C07239=1059.331,223.507,-90.302,172.650,33.223,156.173
C07240=1059.324,223.257,-90.275,172.647,33.219,156.173
C07241=1059.319,223.009,-90.249,172.645,33.215,156.172
C07242=1059.313,222.761,-90.222,172.642,33.212,156.171
C07243=1059.307,222.526,-90.196,172.640,33.208,156.170
C07244=1059.300,222.291,-90.172,172.638,33.204,156.170
C07245=1059.295,222.056,-90.147,172.637,33.201,156.169
C07246=1059.289,221.821,-90.121,172.635,33.197,156.168
C07247=1059.283,221.586,-90.096,172.633,33.193,156.168
C07248=1059.278,221.351,-90.071,172.631,33.190,156.167
C07249=1059.272,221.116,-90.045,172.629,33.185,156.166
C07250=1059.266,220.881,-90.020,172.627,33.182,156.166
C07251=1059.260,220.633,-89.994,172.625,33.178,156.165
C07252=1059.254,220.384,-89.968,172.623,33.174,156.164
C07253=1059.247,220.135,-89.942,172.621,33.171,156.163
C07254=1059.241,219.887,-89.915,172.619,33.166,156.163
C07255=1059.235,219.639,-89.889,172.617,33.163,156.162
C07256=1059.229,219.390,-89.862,172.615,33.159,156.161
C07257=1059.222,219.141,-89.837,172.613,33.155,156.160
C07258=1059.216,218.893,-89.810,172.611,33.151,156.160
C07259=1059.211,218.644,-89.783,172.609,33.147,156.159
C07260=1059.204,218.396,-89.757,172.607,33.143,156.158
C07261=1059.198,218.147,-89.730,172.604,33.140,156.158
C07262=1059.191,217.898,-89.705,172.602,33.135,156.157
C07263=1059.186,217.650,-89.678,172.600,33.132,156.156
C07264=1059.179,217.402,-89.652,172.598,33.128,156.155
C07265=1059.173,217.152,-89.626,172.596,33.124,156.155
C07266=1059.167,216.904,-89.600,172.594,33.120,156.154
C07267=1059.161,216.656,-89.573,172.592,33.116,156.153
C07268=1059.155,216.407,-89.548,172.590,33.112,156.152
C07269=1059.149,216.159,-89.521,172.588,33.108,156.152
C07270=1059.142,215.910,-89.495,172.586,33.104,156.151
C07271=1059.136,215.661,-89.469,172.584,33.101,156.150
C07272=1059.130,215.413,-89.443,172.582,33.096,156.149
C07273=1059.124,215.165,-89.416,172.580,33.093,156.149
C07274=1059.118,214.916,-89.391,172.578,33.088,156.148
C07275=1059.111,214.667,-89.364,172.576,33.085,156.147
C07276=1059.105,214.418,-89.339,172.574,33.080,156.146
C07277=1059.099,214.170,-89.312,172.573,33.077,156.146
C07278=1059.093,213.921,-89.287,172.571,33.073,156.145
C07279=1059.087,213.673,-89.260,172.568,33.069,156.144
C07280=1059.081,213.425,-89.234,172.566,33.065,156.144
C07281=1059.075,213.176,-89.208,172.564,33.061,156.143
C07282=1059.069,212.928,-89.182,172.562,33.057,156.142
C07283=1059.063,212.678,-89.156,172.560,33.053,156.141
C07284=1059.056,212.430,-89.130,172.558,33.049,156.141
C07285=1059.050,212.181,-89.104,172.556,33.045,156.140
C07286=1059.045,211.932,-89.078,172.554,33.041,156.139
C07287=1059.038,211.684,-89.052,172.552,33.037,156.138
C07288=1059.032,211.436,-89.027,172.550,33.033,156.138
C07289=1059.026,211.187,-89.000,172.548,33.029,156.137
C07290=1059.020,210.939,-88.975,172.546,33.026,156.136
C07291=1059.013,210.690,-88.949,172.544,33.022,156.135
C07292=1059.007,210.441,-88.923,172.542,33.018,156.135
C07293=1059.001,210.192,-88.897,172.540,33.014,156.134
C07294=1058.995,209.944,-88.871,172.538,33.010,156.133
C07295=1058.988,209.696,-88.846,172.536,33.006,156.132
C07296=1058.983,209.447,-88.820,172.534,33.002,156.132
C07297=1058.976,209.199,-88.794,172.532,32.998,156.131
C07298=1058.970,208.950,-88.769,172.530,32.994,156.130
C07299=1058.965,208.717,-88.744,172.529,32.990,156.130
C07300=1058.959,208.484,-88.720,172.527,32.986,156.129
C07301=1058.954,208.252,-88.696,172.525,32.983,156.128
C07302=1058.947,208.020,-88.672,172.523,32.979,156.127
C07303=1058.941,207.788,-88.648,172.521,32.975,156.127
C07304=1058.936,207.555,-88.624,172.520,32.972,156.126
C07305=1058.930,207.323,-88.600,172.518,32.968,156.125
C07306=1058.924,207.090,-88.576,172.516,32.964,156.125
C07307=1058.899,206.041,-88.472,172.330,32.878,156.114
C07308=1058.893,205.792,-88.447,172.327,32.874,156.114
C07309=1058.888,205.543,-88.423,172.325,32.871,156.113
C07310=1058.881,205.295,-88.398,172.323,32.868,156.113
C07311=1058.875,205.045,-88.373,172.320,32.865,156.112
C07312=1058.870,204.797,-88.348,172.318,32.862,156.112
C07313=1058.864,204.548,-88.323,172.316,32.859,156.111
C07314=1058.858,204.300,-88.298,172.313,32.856,156.110
C07315=1058.852,204.051,-88.274,172.311,32.853,156.110
C07316=1058.846,203.802,-88.250,172.309,32.850,156.109
C07317=1058.840,203.554,-88.225,172.306,32.846,156.109
C07318=1058.834,203.304,-88.200,172.304,32.843,156.108
C07319=1058.829,203.056,-88.176,172.302,32.841,156.108
C07320=1058.823,202.807,-88.151,172.299,32.838,156.107
C07321=1058.817,202.559,-88.126,172.297,32.834,156.107
C07322=1058.811,202.310,-88.102,172.295,32.831,156.106
C07323=1058.805,202.062,-88.077,172.292,32.828,156.106
C07324=1058.799,201.812,-88.053,172.290,32.825,156.105
C07325=1058.793,201.563,-88.028,172.288,32.822,156.105
C07326=1058.787,201.315,-88.004,172.285,32.819,156.104
C07327=1058.781,201.066,-87.980,172.283,32.816,156.104
C07328=1058.775,200.818,-87.955,172.281,32.813,156.103
C07329=1058.769,200.569,-87.931,172.278,32.810,156.103
C07330=1058.763,200.320,-87.907,172.276,32.807,156.102
C07331=1058.757,200.071,-87.883,172.274,32.804,156.102
C07332=1058.751,199.822,-87.858,172.271,32.801,156.101
C07333=1058.745,199.573,-87.834,172.269,32.798,156.100
C07334=1058.739,199.325,-87.809,172.267,32.796,156.100
C07335=1058.733,199.077,-87.785,172.265,32.792,156.099
C07336=1058.727,198.827,-87.761,172.262,32.789,156.099
C07337=1058.721,198.579,-87.737,172.260,32.787,156.098
C07338=1058.715,198.330,-87.712,172.258,32.783,156.098
C07339=1058.709,198.081,-87.689,172.255,32.780,156.097
C07340=1058.703,197.832,-87.664,172.253,32.778,156.097
C07341=1058.697,197.584,-87.640,172.251,32.775,156.096
C07342=1058.691,197.335,-87.616,172.248,32.771,156.096
C07343=1058.685,197.086,-87.592,172.247,32.769,156.095
C07344=1058.679,196.837,-87.568,172.245,32.766,156.095
C07345=1058.674,196.588,-87.543,172.243,32.762,156.094
C07346=1058.668,196.339,-87.519,172.240,32.760,156.094
C07347=1058.662,196.091,-87.495,172.238,32.757,156.093
C07348=1058.656,195.843,-87.471,172.236,32.754,156.093
C07349=1058.650,195.593,-87.447,172.234,32.751,156.092
C07350=1058.644,195.345,-87.423,172.231,32.748,156.092
C07351=1058.638,195.096,-87.398,172.229,32.745,156.091
C07352=1058.632,194.847,-87.375,172.227,32.742,156.091
C07353=1058.626,194.598,-87.350,172.224,32.739,156.090
C07354=1058.620,194.350,-87.326,172.222,32.736,156.090
C07355=1058.615,194.101,-87.302,172.220,32.733,156.089
C07356=1058.608,193.852,-87.278,172.218,32.730,156.089
C07357=1058.603,193.604,-87.254,172.215,32.727,156.088
C07358=1058.597,193.355,-87.230,172.213,32.724,156.088
C07359=1058.592,193.106,-87.206,172.211,32.722,156.087
C07360=1058.586,192.857,-87.183,172.209,32.718,156.087
C07361=1058.579,192.608,-87.159,172.207,32.715,156.086
C07362=1058.574,192.360,-87.134,172.204,32.713,156.086
C07363=1058.568,192.111,-87.111,172.202,32.709,156.085
C07364=1058.562,191.862,-87.086,172.200,32.707,156.085
C07365=1058.556,191.613,-87.063,172.198,32.704,156.084
C07366=1058.551,191.365,-87.039,172.195,32.700,156.084
C07367=1058.544,191.116,-87.015,172.193,32.698,156.083
C07368=1058.538,190.832,-86.988,172.191,32.695,156.083
C07369=1058.531,190.548,-86.960,172.188,32.691,156.082
C07370=1058.525,190.265,-86.934,172.186,32.688,156.081
C07371=1058.518,189.981,-86.906,172.184,32.684,156.081
C07372=1058.511,189.732,-86.882,172.182,32.681,156.080
C07373=1058.507,189.483,-86.858,172.180,32.679,156.080
C07374=1058.500,189.235,-86.835,172.177,32.675,156.079
C07375=1058.494,188.986,-86.811,172.175,32.672,156.079
C07376=1058.489,188.736,-86.787,172.173,32.670,156.078
C07377=1058.483,188.488,-86.763,172.171,32.667,156.078
C07378=1058.478,188.240,-86.739,172.169,32.664,156.077
C07379=1058.471,187.990,-86.716,172.166,32.661,156.077
C07380=1058.466,187.741,-86.692,172.164,32.658,156.076
C07381=1058.460,187.493,-86.668,172.162,32.655,156.076
C07382=1058.454,187.244,-86.645,172.160,32.652,156.075
C07383=1058.449,186.996,-86.621,172.158,32.649,156.075
C07384=1058.442,186.746,-86.597,172.156,32.646,156.074
C07385=1058.437,186.497,-86.573,172.153,32.644,156.074
C07386=1058.431,186.249,-86.550,172.151,32.640,156.073
C07387=1058.425,186.000,-86.527,172.149,32.638,156.073
C07388=1058.420,185.752,-86.502,172.147,32.635,156.072
C07389=1058.414,185.502,-86.479,172.145,32.631,156.072
C07390=1058.408,185.253,-86.455,172.143,32.629,156.071
C07391=1058.403,185.005,-86.432,172.140,32.626,156.071
C07392=1058.397,184.756,-86.408,172.138,32.623,156.070
C07393=1058.392,184.507,-86.385,172.136,32.620,156.070
C07394=1058.385,184.258,-86.361,172.134,32.617,156.069
C07395=1058.379,184.009,-86.338,172.133,32.614,156.069
C07396=1058.373,183.761,-86.314,172.131,32.612,156.068
C07397=1058.367,183.511,-86.291,172.128,32.609,156.068
C07398=1058.361,183.262,-86.268,172.126,32.606,156.068
C07399=1058.355,183.014,-86.244,172.124,32.603,156.067
C07400=1058.349,182.765,-86.221,172.122,32.601,156.067
C07401=1058.343,182.516,-86.198,172.120,32.598,156.066
C07402=1058.336,182.268,-86.175,172.118,32.595,156.066
C07403=1058.331,182.019,-86.152,172.115,32.592,156.065
C07404=1058.325,181.770,-86.129,172.113,32.590,156.065
C07405=1058.318,181.521,-86.105,172.111,32.587,156.064
C07406=1058.313,181.272,-86.082,172.109,32.584,156.064
C07407=1058.307,181.023,-86.059,172.107,32.581,156.063
C07408=1058.301,180.775,-86.035,172.105,32.579,156.063
C07409=1058.294,180.525,-86.012,172.102,32.576,156.063
C07410=1058.289,180.276,-85.989,172.100,32.573,156.062
C07411=1058.283,180.027,-85.966,172.098,32.570,156.062
C07412=1058.276,179.779,-85.943,172.096,32.568,156.061
C07413=1058.270,179.531,-85.920,172.094,32.565,156.061
C07414=1058.264,179.281,-85.897,172.092,32.562,156.060
C07415=1058.258,179.032,-85.874,172.090,32.559,156.060
C07416=1058.252,178.784,-85.850,172.088,32.557,156.059
C07417=1058.247,178.535,-85.827,172.086,32.554,156.059
C07418=1058.241,178.286,-85.804,172.084,32.551,156.058
C07419=1058.235,178.037,-85.781,172.082,32.548,156.058
C07420=1058.228,177.788,-85.759,172.080,32.546,156.057
C07421=1058.222,177.539,-85.736,172.078,32.543,156.057
C07422=1058.216,177.291,-85.712,172.076,32.540,156.056
C07423=1058.211,177.042,-85.689,172.073,32.537,156.056
C07424=1058.205,176.793,-85.666,172.071,32.535,156.056
C07425=1058.199,176.544,-85.643,172.069,32.532,156.055
C07426=1058.193,176.295,-85.620,172.067,32.529,156.055
C07427=1058.186,176.046,-85.597,172.065,32.527,156.054
C07428=1058.181,175.797,-85.574,172.063,32.524,156.054
C07429=1058.175,175.548,-85.552,172.061,32.521,156.053
C07430=1058.169,175.299,-85.529,172.059,32.518,156.053
C07431=1058.163,175.050,-85.506,172.057,32.516,156.052
C07432=1058.156,174.766,-85.479,172.054,32.512,156.052
C07433=1058.149,174.482,-85.454,172.052,32.509,156.051
C07434=1058.143,174.198,-85.427,172.050,32.506,156.051
C07435=1058.137,173.914,-85.401,172.048,32.503,156.050
C07436=1058.131,173.665,-85.378,172.046,32.500,156.050
C07437=1058.125,173.416,-85.355,172.044,32.498,156.049
C07438=1058.118,173.167,-85.333,172.042,32.495,156.049
C07439=1058.112,172.918,-85.310,172.040,32.492,156.048
C07440=1058.107,172.669,-85.287,172.038,32.489,156.048
C07441=1058.101,172.420,-85.264,172.036,32.487,156.047
C07442=1058.095,172.171,-85.241,172.034,32.483,156.047
C07443=1058.089,171.923,-85.219,172.031,32.481,156.047
C07444=1058.083,171.674,-85.196,172.029,32.478,156.046
C07445=1058.077,171.425,-85.173,172.027,32.476,156.046
C07446=1058.071,171.176,-85.150,172.025,32.472,156.045
C07447=1058.066,170.927,-85.127,172.023,32.470,156.045
C07448=1058.059,170.679,-85.104,172.021,32.467,156.044
C07449=1058.054,170.429,-85.082,172.019,32.465,156.044
C07450=1058.048,170.180,-85.059,172.017,32.461,156.043
C07451=1058.042,169.931,-85.036,172.015,32.459,156.043
C07452=1058.037,169.682,-85.013,172.014,32.456,156.042
C07453=1058.031,169.435,-84.991,172.012,32.454,156.042
C07454=1058.025,169.186,-84.968,172.010,32.451,156.041
C07455=1058.020,168.936,-84.946,172.008,32.448,156.041
C07456=1058.014,168.687,-84.923,172.006,32.445,156.041
C07457=1058.007,168.439,-84.901,172.004,32.443,156.040
C07458=1058.002,168.190,-84.878,172.002,32.440,156.040
C07459=1057.996,167.941,-84.855,172.000,32.437,156.039
C07460=1057.991,167.691,-84.833,171.998,32.434,156.039
C07461=1057.985,167.442,-84.810,171.996,32.432,156.038
C07462=1057.978,167.194,-84.787,171.994,32.429,156.038
C07463=1057.973,166.945,-84.765,171.992,32.426,156.037
C07464=1057.967,166.695,-84.742,171.989,32.423,156.037
C07465=1057.962,166.447,-84.720,171.987,32.421,156.036
C07466=1057.956,166.199,-84.697,171.985,32.418,156.036
C07467=1057.950,165.949,-84.675,171.983,32.415,156.036
C07468=1057.944,165.700,-84.652,171.982,32.412,156.035
C07469=1057.938,165.452,-84.630,171.980,32.410,156.035
C07470=1057.933,165.202,-84.608,171.978,32.407,156.034
C07471=1057.927,164.953,-84.585,171.976,32.404,156.034
C07472=1057.921,164.704,-84.562,171.974,32.401,156.033
C07473=1057.916,164.456,-84.540,171.972,32.399,156.033
C07474=1057.910,164.207,-84.517,171.970,32.396,156.032
C07475=1057.904,163.958,-84.495,171.968,32.393,156.032
C07476=1057.899,163.709,-84.472,171.966,32.391,156.031
C07477=1057.892,163.460,-84.450,171.964,32.388,156.031
C07478=1057.887,163.212,-84.427,171.962,32.385,156.030
C07479=1057.882,162.962,-84.405,171.960,32.382,156.030
C07480=1057.875,162.714,-84.383,171.958,32.380,156.030
C07481=1057.870,162.464,-84.361,171.956,32.376,156.029
C07482=1057.864,162.215,-84.338,171.954,32.374,156.029
C07483=1057.859,161.966,-84.316,171.952,32.371,156.028
C07484=1057.853,161.718,-84.293,171.952,32.369,156.028
C07485=1057.847,161.468,-84.271,171.950,32.366,156.027
C07486=1057.842,161.219,-84.248,171.948,32.363,156.027
C07487=1057.835,160.970,-84.227,171.946,32.360,156.026
C07488=1057.830,160.722,-84.204,171.944,32.358,156.026
C07489=1057.824,160.473,-84.182,171.942,32.355,156.025
C07490=1057.818,160.224,-84.159,171.940,32.353,156.025
C07491=1057.812,159.975,-84.138,171.938,32.350,156.025
C07492=1057.806,159.726,-84.115,171.936,32.347,156.024
C07493=1057.800,159.477,-84.093,171.934,32.344,156.024
C07494=1057.795,159.228,-84.072,171.932,32.342,156.023
C07495=1057.788,158.980,-84.050,171.930,32.339,156.023
C07496=1057.782,158.694,-84.025,171.927,32.336,156.022
C07497=1057.775,158.410,-83.999,171.925,32.333,156.022
C07498=1057.768,158.126,-83.973,171.924,32.330,156.021
C07499=1057.762,157.841,-83.949,171.922,32.327,156.021
C07500=1057.756,157.592,-83.927,171.920,32.325,156.020
C07501=1057.749,157.343,-83.905,171.918,32.322,156.020
C07502=1057.744,157.094,-83.882,171.916,32.319,156.020
C07503=1057.738,156.845,-83.861,171.914,32.317,156.019
C07504=1057.732,156.597,-83.839,171.912,32.314,156.019
C07505=1057.726,156.347,-83.817,171.910,32.311,156.018
C07506=1057.720,156.098,-83.795,171.908,32.309,156.018
C07507=1057.714,155.849,-83.773,171.906,32.306,156.017
C07508=1057.709,155.601,-83.751,171.904,32.303,156.017
C07509=1057.703,155.351,-83.729,171.902,32.301,156.016
C07510=1057.697,155.102,-83.707,171.900,32.298,156.016
C07511=1057.691,154.853,-83.686,171.898,32.296,156.016
C07512=1057.685,154.605,-83.663,171.897,32.293,156.015
C07513=1057.679,154.356,-83.642,171.895,32.290,156.015
C07514=1057.673,154.106,-83.620,171.893,32.288,156.014
C07515=1057.667,153.857,-83.598,171.891,32.285,156.014
C07516=1057.661,153.609,-83.577,171.889,32.282,156.013
C07517=1057.656,153.360,-83.554,171.887,32.280,156.013
C07518=1057.649,153.111,-83.533,171.885,32.277,156.013
C07519=1057.643,152.861,-83.511,171.883,32.275,156.012
C07520=1057.638,152.613,-83.490,171.882,32.272,156.012
C07521=1057.632,152.364,-83.468,171.880,32.270,156.011
C07522=1057.625,152.114,-83.446,171.878,32.267,156.011
C07523=1057.620,151.865,-83.424,171.876,32.264,156.010
C07524=1057.614,151.616,-83.403,171.874,32.262,156.010
C07525=1057.608,151.368,-83.380,171.872,32.259,156.010
C07526=1057.602,151.119,-83.359,171.871,32.257,156.009
C07527=1057.596,150.870,-83.338,171.869,32.254,156.009
C07528=1057.590,150.621,-83.316,171.867,32.251,156.008
C07529=1057.585,150.371,-83.294,171.865,32.249,156.008
C07530=1057.579,150.123,-83.272,171.863,32.246,156.007
C07531=1057.573,149.874,-83.251,171.861,32.244,156.007
C07532=1057.567,149.625,-83.229,171.859,32.241,156.007
C07533=1057.561,149.376,-83.208,171.857,32.238,156.006
C07534=1057.555,149.127,-83.186,171.856,32.236,156.006
C07535=1057.549,148.878,-83.165,171.854,32.233,156.005
C07536=1057.543,148.629,-83.143,171.852,32.231,156.005
C07537=1057.537,148.380,-83.122,171.850,32.228,156.004
C07538=1057.531,148.131,-83.100,171.848,32.225,156.004
C07539=1057.526,147.882,-83.078,171.846,32.223,156.004
C07540=1057.520,147.633,-83.057,171.845,32.220,156.003
C07541=1057.514,147.383,-83.035,171.843,32.218,156.003
C07542=1057.508,147.135,-83.014,171.841,32.215,156.002
C07543=1057.502,146.885,-82.993,171.839,32.212,156.002
C07544=1057.495,146.636,-82.972,171.837,32.210,156.002
C07545=1057.490,146.388,-82.950,171.835,32.207,156.001
C07546=1057.484,146.139,-82.929,171.834,32.205,156.001
C07547=1057.478,145.890,-82.908,171.832,32.202,156.000
C07548=1057.472,145.641,-82.886,171.830,32.199,156.000
C07549=1057.466,145.392,-82.864,171.828,32.197,155.999
C07550=1057.460,145.143,-82.843,171.826,32.195,155.999
C07551=1057.454,144.893,-82.822,171.824,32.192,155.999
C07552=1057.448,144.644,-82.800,171.823,32.190,155.998
C07553=1057.443,144.396,-82.779,171.821,32.187,155.998
C07554=1057.437,144.146,-82.758,171.819,32.184,155.997
C07555=1057.431,143.898,-82.736,171.817,32.182,155.997
C07556=1057.424,143.648,-82.716,171.816,32.179,155.997
C07557=1057.418,143.399,-82.694,171.814,32.177,155.996
C07558=1057.413,143.151,-82.673,171.812,32.174,155.996
C07559=1057.407,142.901,-82.651,171.810,32.171,155.995
C07560=1057.401,142.616,-82.628,171.808,32.169,155.995
C07561=1057.394,142.332,-82.603,171.806,32.166,155.994
C07562=1057.386,142.047,-82.579,171.803,32.163,155.994
C07563=1057.380,141.763,-82.554,171.801,32.160,155.993
C07564=1057.374,141.513,-82.533,171.800,32.157,155.993
C07565=1057.368,141.265,-82.513,171.799,32.155,155.992
C07566=1057.362,141.015,-82.491,171.797,32.152,155.992
C07567=1057.356,140.766,-82.470,171.795,32.149,155.992
C07568=1057.351,140.517,-82.449,171.793,32.147,155.991
C07569=1057.344,140.268,-82.427,171.791,32.144,155.991
C07570=1057.339,140.019,-82.407,171.789,32.142,155.990
C07571=1057.333,139.769,-82.385,171.787,32.139,155.990
C07572=1057.327,139.521,-82.364,171.786,32.137,155.990
C07573=1057.321,139.271,-82.343,171.784,32.134,155.989
C07574=1057.315,139.023,-82.322,171.782,32.132,155.989
C07575=1057.309,138.773,-82.301,171.780,32.129,155.988
C07576=1057.303,138.525,-82.281,171.778,32.126,155.988
C07577=1057.297,138.276,-82.259,171.777,32.124,155.987
C07578=1057.292,138.027,-82.238,171.775,32.121,155.987
C07579=1057.285,137.777,-82.217,171.773,32.119,155.987
C07580=1057.279,137.529,-82.197,171.772,32.117,155.986
C07581=1057.273,137.279,-82.175,171.770,32.114,155.986
C07582=1057.268,137.030,-82.155,171.768,32.111,155.985
C07583=1057.261,136.781,-82.133,171.766,32.109,155.985
C07584=1057.256,136.532,-82.113,171.764,32.106,155.985
C07585=1057.250,136.283,-82.091,171.762,32.104,155.984
C07586=1057.244,136.034,-82.071,171.760,32.102,155.984
C07587=1057.238,135.785,-82.050,171.759,32.099,155.983
C07588=1057.232,135.536,-82.029,171.757,32.096,155.983
C07589=1057.225,135.287,-82.008,171.756,32.094,155.983
C07590=1057.220,135.038,-81.988,171.754,32.091,155.982
C07591=1057.214,134.789,-81.966,171.752,32.089,155.982
C07592=1057.208,134.540,-81.946,171.750,32.086,155.981
C07593=1057.202,134.291,-81.924,171.749,32.084,155.981
C07594=1057.196,134.042,-81.904,171.747,32.081,155.981
C07595=1057.190,133.792,-81.883,171.745,32.079,155.980
C07596=1057.184,133.543,-81.862,171.743,32.076,155.980
C07597=1057.178,133.295,-81.842,171.741,32.074,155.979
C07598=1057.172,133.045,-81.821,171.739,32.071,155.979
C07599=1057.167,132.796,-81.800,171.738,32.068,155.978
C07600=1057.160,132.547,-81.780,171.737,32.066,155.978
C07601=1057.155,132.298,-81.758,171.735,32.063,155.978
C07602=1057.149,132.050,-81.738,171.733,32.061,155.977
C07603=1057.143,131.800,-81.718,171.731,32.059,155.977
C07604=1057.137,131.551,-81.696,171.729,32.056,155.976
C07605=1057.131,131.302,-81.676,171.728,32.053,155.976
C07606=1057.125,131.053,-81.656,171.726,32.051,155.976
C07607=1057.119,130.804,-81.634,171.724,32.049,155.975
C07608=1057.113,130.555,-81.614,171.722,32.046,155.975
C07609=1057.106,130.305,-81.594,171.720,32.044,155.974
C07610=1057.101,130.056,-81.574,171.718,32.041,155.974
C07611=1057.094,129.807,-81.552,171.717,32.039,155.974
C07612=1057.089,129.558,-81.532,171.716,32.036,155.973
C07613=1057.083,129.309,-81.512,171.714,32.034,155.973
C07614=1057.076,129.060,-81.492,171.712,32.031,155.972
C07615=1057.071,128.811,-81.470,171.710,32.029,155.972
C07616=1057.064,128.562,-81.450,171.708,32.026,155.972
C07617=1057.058,128.313,-81.430,171.707,32.024,155.971
C07618=1057.053,128.064,-81.410,171.705,32.021,155.971
C07619=1057.046,127.814,-81.389,171.703,32.019,155.971
C07620=1057.040,127.566,-81.369,171.701,32.017,155.970
C07621=1057.034,127.316,-81.348,171.699,32.014,155.970
C07622=1057.028,127.068,-81.328,171.698,32.012,155.969
C07623=1057.022,126.819,-81.308,171.697,32.010,155.969
C07624=1057.015,126.533,-81.284,171.695,32.006,155.968
C07625=1057.009,126.249,-81.261,171.693,32.004,155.968
C07626=1057.002,125.963,-81.237,171.690,32.001,155.968
C07627=1056.994,125.679,-81.214,171.688,31.998,155.967
C07628=1056.989,125.429,-81.194,171.687,31.996,155.967
C07629=1056.983,125.180,-81.174,171.685,31.993,155.966
C07630=1056.977,124.931,-81.154,171.683,31.991,155.966
C07631=1056.971,124.682,-81.133,171.681,31.988,155.965
C07632=1056.965,124.433,-81.113,171.679,31.986,155.965
C07633=1056.959,124.184,-81.093,171.679,31.983,155.965
C07634=1056.952,123.935,-81.072,171.677,31.981,155.964
C07635=1056.947,123.685,-81.052,171.675,31.978,155.964
C07636=1056.941,123.437,-81.032,171.673,31.975,155.963
C07637=1056.934,123.187,-81.012,171.671,31.973,155.963
C07638=1056.929,122.938,-80.991,171.670,31.971,155.963
C07639=1056.923,122.689,-80.971,171.668,31.968,155.962
C07640=1056.916,122.440,-80.951,171.666,31.966,155.962
C07641=1056.911,122.190,-80.930,171.664,31.963,155.961
C07642=1056.905,121.942,-80.910,171.662,31.961,155.961
C07643=1056.899,121.693,-80.890,171.661,31.958,155.961
C07644=1056.893,121.443,-80.870,171.660,31.956,155.960
C07645=1056.887,121.194,-80.849,171.658,31.953,155.960
C07646=1056.881,120.945,-80.829,171.656,31.951,155.959
C07647=1056.875,120.697,-80.809,171.655,31.949,155.959
C07648=1056.869,120.447,-80.789,171.653,31.946,155.959
C07649=1056.863,120.198,-80.769,171.651,31.943,155.958
C07650=1056.857,119.949,-80.749,171.649,31.941,155.958
C07651=1056.851,119.700,-80.729,171.647,31.938,155.957
C07652=1056.846,119.450,-80.708,171.646,31.936,155.957
C07653=1056.840,119.202,-80.688,171.644,31.934,155.957
C07654=1056.834,118.952,-80.669,171.643,31.931,155.956
C07655=1056.828,118.703,-80.649,171.641,31.928,155.956
C07656=1056.822,118.454,-80.628,171.640,31.926,155.955
C07657=1056.816,118.205,-80.608,171.638,31.923,155.955
C07658=1056.810,117.956,-80.588,171.636,31.921,155.955
C07659=1056.804,117.707,-80.568,171.634,31.918,155.954
C07660=1056.799,117.458,-80.547,171.633,31.916,155.954
C07661=1056.793,117.209,-80.528,171.631,31.913,155.953
C07662=1056.787,116.959,-80.508,171.629,31.911,155.953
C07663=1056.781,116.710,-80.488,171.627,31.908,155.953
C07664=1056.775,116.461,-80.468,171.626,31.906,155.952
C07665=1056.769,116.212,-80.447,171.625,31.904,155.952
C07666=1056.764,115.963,-80.428,171.623,31.901,155.951
C07667=1056.758,115.714,-80.408,171.621,31.898,155.951
C07668=1056.751,115.465,-80.388,171.620,31.896,155.951
C07669=1056.746,115.215,-80.367,171.618,31.893,155.950
C07670=1056.740,114.966,-80.348,171.616,31.891,155.950
C07671=1056.734,114.717,-80.328,171.614,31.888,155.949
C07672=1056.728,114.468,-80.308,171.613,31.886,155.949
C07673=1056.723,114.219,-80.287,171.611,31.883,155.949
C07674=1056.717,113.970,-80.268,171.610,31.881,155.948
C07675=1056.711,113.720,-80.248,171.608,31.878,155.948
C07676=1056.705,113.472,-80.228,171.606,31.876,155.947
C07677=1056.699,113.222,-80.209,171.605,31.873,155.947
C07678=1056.693,112.973,-80.189,171.603,31.871,155.947
C07679=1056.687,112.724,-80.169,171.601,31.869,155.946
C07680=1056.681,112.475,-80.149,171.599,31.866,155.946
C07681=1056.675,112.226,-80.129,171.598,31.864,155.945
C07682=1056.669,111.977,-80.109,171.596,31.861,155.945
C07683=1056.663,111.727,-80.090,171.594,31.859,155.945
C07684=1056.657,111.478,-80.070,171.593,31.856,155.944
C07685=1056.651,111.229,-80.051,171.592,31.854,155.944
C07686=1056.645,110.980,-80.031,171.590,31.851,155.943
C07687=1056.638,110.730,-80.012,171.588,31.849,155.943
C07688=1056.632,110.446,-79.988,171.586,31.846,155.943
C07689=1056.625,110.161,-79.967,171.584,31.843,155.942
C07690=1056.618,109.876,-79.945,171.582,31.841,155.942
C07691=1056.610,109.591,-79.921,171.580,31.838,155.941
C07692=1056.605,109.341,-79.902,171.578,31.835,155.941
C07693=1056.599,109.092,-79.882,171.577,31.833,155.941
C07694=1056.593,108.843,-79.863,171.576,31.831,155.940
C07695=1056.587,108.594,-79.843,171.574,31.828,155.940
C07696=1056.581,108.345,-79.824,171.572,31.825,155.939
C07697=1056.575,108.096,-79.804,171.571,31.823,155.939
C07698=1056.569,107.847,-79.785,171.569,31.821,155.939
C07699=1056.562,107.597,-79.765,171.567,31.818,155.938
C07700=1056.557,107.348,-79.746,171.565,31.816,155.938
C07701=1056.551,107.098,-79.726,171.564,31.814,155.937
C07702=1056.544,106.850,-79.707,171.562,31.811,155.937
C07703=1056.539,106.600,-79.688,171.561,31.809,155.937
C07704=1056.533,106.352,-79.668,171.560,31.806,155.936
C07705=1056.527,106.102,-79.649,171.558,31.804,155.936
C07706=1056.521,105.853,-79.629,171.556,31.801,155.935
C07707=1056.514,105.604,-79.610,171.554,31.799,155.935
C07708=1056.509,105.355,-79.591,171.553,31.797,155.935
C07709=1056.503,105.106,-79.571,171.551,31.794,155.934
C07710=1056.497,104.857,-79.552,171.549,31.792,155.934
C07711=1056.491,104.607,-79.532,171.547,31.789,155.934
C07712=1056.485,104.359,-79.513,171.546,31.787,155.933
C07713=1056.478,104.109,-79.493,171.545,31.784,155.933
C07714=1056.473,103.859,-79.474,171.543,31.782,155.932
C07715=1056.467,103.610,-79.454,171.541,31.779,155.932
C07716=1056.461,103.361,-79.435,171.540,31.777,155.932
C07717=1056.455,103.112,-79.416,171.538,31.775,155.931
C07718=1056.449,102.863,-79.396,171.536,31.772,155.931
C07719=1056.443,102.613,-79.377,171.535,31.770,155.930
C07720=1056.437,102.364,-79.358,171.533,31.767,155.930
C07721=1056.431,102.115,-79.338,171.531,31.765,155.930
C07722=1056.425,101.866,-79.319,171.530,31.762,155.929
C07723=1056.419,101.617,-79.300,171.529,31.760,155.929
C07724=1056.413,101.367,-79.281,171.527,31.757,155.928
C07725=1056.407,101.118,-79.261,171.525,31.755,155.928
C07726=1056.401,100.869,-79.242,171.524,31.752,155.928
C07727=1056.395,100.620,-79.223,171.522,31.750,155.927
C07728=1056.390,100.370,-79.204,171.520,31.748,155.927
C07729=1056.383,100.122,-79.184,171.518,31.745,155.927
C07730=1056.377,99.873,-79.165,171.517,31.743,155.926
C07731=1056.371,99.623,-79.146,171.516,31.741,155.926
C07732=1056.365,99.374,-79.127,171.514,31.738,155.925
C07733=1056.359,99.125,-79.108,171.513,31.736,155.925
C07734=1056.353,98.875,-79.089,171.511,31.733,155.925
C07735=1056.347,98.626,-79.071,171.509,31.731,155.924
C07736=1056.341,98.377,-79.051,171.507,31.729,155.924
C07737=1056.334,98.128,-79.032,171.506,31.726,155.924
C07738=1056.328,97.879,-79.013,171.504,31.723,155.923
C07739=1056.323,97.629,-78.993,171.502,31.721,155.923
C07740=1056.316,97.380,-78.975,171.501,31.719,155.922
C07741=1056.311,97.131,-78.956,171.500,31.716,155.922
C07742=1056.305,96.883,-78.937,171.498,31.714,155.922
C07743=1056.299,96.633,-78.918,171.496,31.711,155.921
C07744=1056.293,96.384,-78.899,171.495,31.710,155.921
C07745=1056.287,96.135,-78.880,171.493,31.707,155.921
C07746=1056.280,95.886,-78.861,171.491,31.704,155.920
C07747=1056.275,95.637,-78.842,171.489,31.702,155.920
C07748=1056.268,95.387,-78.823,171.488,31.700,155.919
C07749=1056.262,95.138,-78.804,171.487,31.697,155.919
C07750=1056.256,94.889,-78.785,171.485,31.695,155.919
C07751=1056.250,94.639,-78.766,171.484,31.692,155.918
C07752=1056.244,94.354,-78.745,171.482,31.690,155.918
C07753=1056.236,94.069,-78.723,171.480,31.687,155.917
C07754=1056.229,93.784,-78.701,171.478,31.684,155.917
C07755=1056.223,93.499,-78.679,171.476,31.681,155.916
C07756=1056.216,93.250,-78.661,171.474,31.679,155.916
C07757=1056.211,93.001,-78.642,171.473,31.676,155.916
C07758=1056.205,92.752,-78.624,171.472,31.674,155.915
C07759=1056.199,92.502,-78.604,171.470,31.671,155.915
C07760=1056.193,92.253,-78.586,171.468,31.669,155.915
C07761=1056.187,92.004,-78.567,171.467,31.667,155.914
C07762=1056.181,91.755,-78.548,171.465,31.664,155.914
C07763=1056.175,91.505,-78.529,171.463,31.662,155.913
C07764=1056.169,91.257,-78.510,171.462,31.659,155.913
C07765=1056.164,91.007,-78.491,171.460,31.657,155.913
C07766=1056.157,90.758,-78.473,171.459,31.655,155.912
C07767=1056.151,90.509,-78.453,171.457,31.652,155.912
C07768=1056.145,90.260,-78.435,171.456,31.650,155.911
C07769=1056.139,90.010,-78.417,171.454,31.647,155.911
C07770=1056.132,89.761,-78.398,171.452,31.645,155.911
C07771=1056.127,89.511,-78.379,171.451,31.643,155.910
C07772=1056.120,89.262,-78.360,171.449,31.640,155.910
C07773=1056.114,89.014,-78.342,171.447,31.638,155.910
C07774=1056.108,88.764,-78.324,171.445,31.635,155.909
C07775=1056.103,88.515,-78.305,171.445,31.633,155.909
C07776=1056.096,88.265,-78.286,171.443,31.631,155.909
C07777=1056.090,88.016,-78.267,171.441,31.628,155.908
C07778=1056.083,87.767,-78.249,171.440,31.626,155.908
C07779=1056.078,87.517,-78.230,171.438,31.624,155.907
C07780=1056.072,87.269,-78.212,171.436,31.622,155.907
C07781=1056.066,87.020,-78.193,171.435,31.619,155.907
C07782=1056.059,86.770,-78.175,171.433,31.616,155.906
C07783=1056.053,86.521,-78.157,171.432,31.614,155.906
C07784=1056.048,86.271,-78.137,171.430,31.612,155.906
C07785=1056.041,86.022,-78.119,171.429,31.610,155.905
C07786=1056.036,85.773,-78.101,171.427,31.607,155.905
C07787=1056.029,85.524,-78.083,171.425,31.604,155.904
C07788=1056.023,85.275,-78.063,171.424,31.602,155.904
C07789=1056.017,85.025,-78.045,171.422,31.600,155.904
C07790=1056.011,84.776,-78.027,171.420,31.598,155.903
C07791=1056.005,84.527,-78.008,171.419,31.595,155.903
C07792=1055.999,84.278,-77.990,171.418,31.593,155.903
C07793=1055.993,84.028,-77.971,171.416,31.590,155.902
C07794=1055.987,83.779,-77.953,171.415,31.588,155.902
C07795=1055.981,83.529,-77.935,171.413,31.586,155.902
C07796=1055.975,83.281,-77.916,171.411,31.583,155.901
C07797=1055.969,83.032,-77.898,171.409,31.581,155.901
C07798=1055.962,82.782,-77.880,171.408,31.579,155.900
C07799=1055.957,82.533,-77.861,171.406,31.576,155.900
C07800=1055.951,82.284,-77.842,171.405,31.574,155.900
C07801=1055.945,82.034,-77.824,171.404,31.571,155.899
C07802=1055.938,81.785,-77.806,171.402,31.569,155.899
C07803=1055.932,81.536,-77.788,171.400,31.567,155.899
C07804=1055.927,81.287,-77.769,171.399,31.564,155.898
C07805=1055.921,81.037,-77.751,171.397,31.561,155.898
C07806=1055.915,80.788,-77.732,171.395,31.559,155.897
C07807=1055.909,80.539,-77.714,171.394,31.557,155.897
C07808=1055.903,80.290,-77.696,171.393,31.555,155.897
C07809=1055.896,80.041,-77.677,171.391,31.552,155.896
C07810=1055.891,79.791,-77.659,171.390,31.550,155.896
C07811=1055.885,79.542,-77.641,171.388,31.547,155.896
C07812=1055.879,79.292,-77.623,171.386,31.545,155.895
C07813=1055.872,79.043,-77.604,171.384,31.542,155.895
C07814=1055.867,78.794,-77.587,171.383,31.540,155.894
C07815=1055.861,78.545,-77.568,171.381,31.537,155.894
C07816=1055.853,78.260,-77.547,171.380,31.535,155.894
C07817=1055.847,77.975,-77.526,171.378,31.532,155.893
C07818=1055.840,77.690,-77.506,171.376,31.529,155.893
C07819=1055.833,77.404,-77.485,171.374,31.527,155.892
C07820=1055.827,77.155,-77.467,171.373,31.524,155.892
C07821=1055.821,76.906,-77.449,171.371,31.522,155.892
C07822=1055.815,76.656,-77.431,171.369,31.520,155.891
C07823=1055.808,76.407,-77.412,171.368,31.518,155.891
C07824=1055.803,76.158,-77.395,171.367,31.515,155.890
C07825=1055.797,75.909,-77.377,171.365,31.513,155.890
C07826=1055.790,75.659,-77.358,171.364,31.510,155.890
C07827=1055.785,75.410,-77.340,171.362,31.508,155.889
C07828=1055.779,75.161,-77.323,171.360,31.506,155.889
C07829=1055.772,74.911,-77.304,171.359,31.503,155.889
C07830=1055.766,74.663,-77.287,171.357,31.501,155.888
C07831=1055.760,74.413,-77.269,171.355,31.498,155.888
C07832=1055.753,74.164,-77.250,171.354,31.496,155.888
C07833=1055.748,73.915,-77.233,171.353,31.494,155.887
C07834=1055.742,73.665,-77.215,171.351,31.492,155.887
C07835=1055.735,73.416,-77.196,171.349,31.489,155.886
C07836=1055.730,73.167,-77.179,171.348,31.487,155.886
C07837=1055.724,72.917,-77.161,171.346,31.484,155.886
C07838=1055.718,72.667,-77.143,171.344,31.482,155.885
C07839=1055.712,72.419,-77.124,171.343,31.480,155.885
C07840=1055.706,72.169,-77.107,171.342,31.477,155.885
C07841=1055.699,71.920,-77.089,171.340,31.475,155.884
C07842=1055.693,71.671,-77.072,171.339,31.472,155.884
C07843=1055.687,71.422,-77.053,171.337,31.470,155.884
C07844=1055.681,71.173,-77.035,171.335,31.468,155.883
C07845=1055.675,70.923,-77.017,171.334,31.466,155.883
C07846=1055.669,70.673,-77.000,171.332,31.463,155.882
C07847=1055.663,70.425,-76.981,171.331,31.461,155.882
C07848=1055.656,70.175,-76.964,171.330,31.458,155.882
C07849=1055.651,69.926,-76.946,171.328,31.456,155.881
C07850=1055.645,69.677,-76.928,171.326,31.454,155.881
C07851=1055.639,69.427,-76.911,171.324,31.451,155.881
C07852=1055.633,69.178,-76.893,171.323,31.449,155.880
C07853=1055.626,68.928,-76.876,171.321,31.446,155.880
C07854=1055.620,68.680,-76.857,171.319,31.444,155.880
C07855=1055.614,68.430,-76.839,171.319,31.442,155.879
C07856=1055.608,68.180,-76.821,171.317,31.440,155.879
C07857=1055.602,67.932,-76.804,171.315,31.437,155.878
C07858=1055.596,67.682,-76.787,171.314,31.435,155.878
C07859=1055.590,67.433,-76.769,171.312,31.432,155.878
C07860=1055.583,67.184,-76.752,171.310,31.430,155.877
C07861=1055.578,66.934,-76.734,171.309,31.428,155.877
C07862=1055.572,66.685,-76.716,171.307,31.426,155.877
C07863=1055.566,66.435,-76.698,171.306,31.423,155.876
C07864=1055.559,66.187,-76.681,171.305,31.421,155.876
C07865=1055.553,65.937,-76.663,171.303,31.418,155.876
C07866=1055.547,65.688,-76.645,171.301,31.416,155.875
C07867=1055.541,65.439,-76.628,171.299,31.414,155.875
C07868=1055.535,65.190,-76.610,171.298,31.412,155.875
C07869=1055.529,64.940,-76.592,171.296,31.409,155.874
C07870=1055.523,64.691,-76.575,171.295,31.407,155.874
C07871=1055.517,64.441,-76.557,171.294,31.404,155.873
C07872=1055.510,64.192,-76.539,171.292,31.402,155.873
C07873=1055.504,63.943,-76.522,171.290,31.400,155.873
C07874=1055.498,63.693,-76.504,171.289,31.398,155.872
C07875=1055.492,63.444,-76.488,171.287,31.395,155.872
C07876=1055.485,63.194,-76.471,171.285,31.393,155.872
C07877=1055.480,62.945,-76.453,171.284,31.391,155.871
C07878=1055.473,62.696,-76.436,171.283,31.389,155.871
C07879=1055.467,62.446,-76.418,171.281,31.386,155.871
C07880=1055.459,62.162,-76.398,171.279,31.383,155.870
C07881=1055.452,61.876,-76.378,171.277,31.381,155.870
C07882=1055.446,61.591,-76.359,171.275,31.379,155.870
C07883=1055.438,61.306,-76.339,171.273,31.376,155.869
C07884=1055.432,61.057,-76.321,171.272,31.373,155.869
C07885=1055.426,60.807,-76.305,171.271,31.371,155.868
C07886=1055.420,60.558,-76.288,171.269,31.369,155.868
C07887=1055.414,60.308,-76.270,171.268,31.367,155.868
C07888=1055.407,60.059,-76.252,171.266,31.365,155.867
C07889=1055.401,59.810,-76.235,171.264,31.362,155.867
C07890=1055.394,59.560,-76.217,171.263,31.360,155.867
C07891=1055.388,59.311,-76.201,171.261,31.358,155.866
C07892=1055.382,59.061,-76.183,171.259,31.355,155.866
C07893=1055.376,58.813,-76.166,171.258,31.353,155.866
C07894=1055.370,58.563,-76.148,171.257,31.351,155.865
C07895=1055.364,58.314,-76.131,171.255,31.348,155.865
C07896=1055.358,58.065,-76.115,171.253,31.346,155.865
C07897=1055.352,57.815,-76.097,171.252,31.344,155.864
C07898=1055.345,57.566,-76.080,171.250,31.342,155.864
C07899=1055.339,57.316,-76.062,171.248,31.339,155.864
C07900=1055.333,57.067,-76.046,171.248,31.337,155.863
C07901=1055.326,56.818,-76.029,171.246,31.334,155.863
C07902=1055.321,56.569,-76.011,171.244,31.332,155.863
C07903=1055.314,56.319,-75.994,171.243,31.330,155.862
C07904=1055.309,56.070,-75.977,171.241,31.328,155.862
C07905=1055.302,55.820,-75.960,171.239,31.326,155.862
C07906=1055.296,55.571,-75.943,171.237,31.323,155.861
C07907=1055.290,55.322,-75.926,171.236,31.321,155.861
C07908=1055.284,55.072,-75.908,171.235,31.319,155.861
C07909=1055.277,54.824,-75.891,171.233,31.316,155.860
C07910=1055.271,54.573,-75.874,171.232,31.314,155.860
C07911=1055.265,54.325,-75.857,171.230,31.312,155.859
C07912=1055.259,54.075,-75.839,171.228,31.309,155.859
C07913=1055.253,53.825,-75.823,171.227,31.307,155.859
C07914=1055.247,53.577,-75.806,171.225,31.305,155.858
C07915=1055.241,53.327,-75.788,171.224,31.303,155.858
C07916=1055.235,53.078,-75.772,171.223,31.300,155.858
C07917=1055.229,52.829,-75.755,171.221,31.298,155.857
C07918=1055.222,52.579,-75.737,171.219,31.295,155.857
C07919=1055.216,52.330,-75.721,171.217,31.293,155.857
C07920=1055.210,52.080,-75.703,171.216,31.291,155.856
C07921=1055.204,51.831,-75.686,171.214,31.289,155.856
C07922=1055.198,51.582,-75.670,171.213,31.286,155.856
C07923=1055.192,51.332,-75.653,171.212,31.284,155.855
C07924=1055.186,51.083,-75.635,171.210,31.282,155.855
C07925=1055.180,50.834,-75.618,171.208,31.279,155.855
C07926=1055.173,50.584,-75.602,171.207,31.277,155.854
C07927=1055.168,50.335,-75.584,171.205,31.275,155.854
C07928=1055.162,50.086,-75.568,171.203,31.272,155.854
C07929=1055.155,49.836,-75.551,171.203,31.270,155.853
C07930=1055.150,49.587,-75.534,171.201,31.268,155.853
C07931=1055.143,49.338,-75.517,171.199,31.265,155.852
C07932=1055.137,49.088,-75.500,171.198,31.263,155.852
C07933=1055.131,48.839,-75.483,171.196,31.261,155.852
C07934=1055.125,48.589,-75.466,171.194,31.258,155.851
C07935=1055.119,48.341,-75.449,171.192,31.256,155.851
C07936=1055.113,48.090,-75.432,171.192,31.254,155.851
C07937=1055.107,47.842,-75.415,171.190,31.252,155.850
C07938=1055.101,47.592,-75.399,171.188,31.249,155.850
C07939=1055.094,47.343,-75.382,171.187,31.247,155.850
C07940=1055.089,47.093,-75.365,171.185,31.244,155.849
C07941=1055.083,46.844,-75.348,171.183,31.242,155.849
C07942=1055.077,46.595,-75.331,171.182,31.240,155.849
C07943=1055.071,46.345,-75.314,171.181,31.238,155.848
C07944=1055.064,46.060,-75.295,171.179,31.235,155.848
C07945=1055.058,45.775,-75.276,171.177,31.232,155.847
C07946=1055.050,45.488,-75.257,171.175,31.229,155.847
C07947=1055.044,45.203,-75.237,171.173,31.227,155.847
C07948=1055.038,44.954,-75.221,171.172,31.225,155.846
C07949=1055.031,44.704,-75.204,171.171,31.222,155.846
C07950=1055.026,44.455,-75.187,171.169,31.220,155.846
C07951=1055.020,44.205,-75.171,171.167,31.217,155.845
C07952=1055.014,43.957,-75.154,171.166,31.215,155.845
C07953=1055.007,43.707,-75.137,171.164,31.213,155.845
C07954=1055.002,43.457,-75.120,171.162,31.211,155.844
C07955=1054.996,43.208,-75.103,171.161,31.208,155.844
C07956=1054.990,42.959,-75.087,171.160,31.206,155.844
C07957=1054.983,42.709,-75.070,171.158,31.204,155.843
C07958=1054.977,42.460,-75.053,171.157,31.201,155.843
C07959=1054.971,42.211,-75.037,171.155,31.199,155.843
C07960=1054.965,41.961,-75.021,171.153,31.197,155.842
C07961=1054.958,41.711,-75.004,171.151,31.194,155.842
C07962=1054.952,41.463,-74.987,171.150,31.192,155.842
C07963=1054.946,41.213,-74.971,171.149,31.190,155.841
C07964=1054.940,40.964,-74.955,171.147,31.188,155.841
C07965=1054.934,40.715,-74.939,171.146,31.186,155.840
C07966=1054.928,40.464,-74.922,171.144,31.184,155.840
C07967=1054.921,40.216,-74.905,171.142,31.181,155.840
C07968=1054.916,39.966,-74.889,171.141,31.179,155.839
C07969=1054.910,39.717,-74.872,171.139,31.177,155.839
C07970=1054.904,39.468,-74.856,171.138,31.174,155.839
C07971=1054.897,39.218,-74.840,171.136,31.172,155.839
C07972=1054.891,38.969,-74.823,171.135,31.169,155.838
C07973=1054.885,38.720,-74.806,171.133,31.167,155.838
C07974=1054.879,38.470,-74.790,171.131,31.165,155.838
C07975=1054.874,38.221,-74.773,171.130,31.163,155.837
C07976=1054.868,37.971,-74.757,171.128,31.161,155.837
C07977=1054.861,37.721,-74.740,171.127,31.158,155.837
C07978=1054.855,37.472,-74.725,171.125,31.156,155.836
C07979=1054.849,37.223,-74.708,171.124,31.154,155.836
C07980=1054.842,36.974,-74.692,171.122,31.152,155.835
C07981=1054.836,36.725,-74.675,171.120,31.150,155.835
C07982=1054.830,36.475,-74.659,171.119,31.147,155.835
C07983=1054.824,36.225,-74.642,171.117,31.145,155.834
C07984=1054.817,35.976,-74.627,171.116,31.143,155.834
C07985=1054.811,35.727,-74.610,171.114,31.141,155.834
C07986=1054.805,35.478,-74.594,171.113,31.138,155.833
C07987=1054.799,35.228,-74.578,171.111,31.136,155.833
C07988=1054.793,34.978,-74.561,171.109,31.134,155.833
C07989=1054.787,34.729,-74.545,171.108,31.132,155.833
C07990=1054.780,34.480,-74.529,171.107,31.129,155.832
C07991=1054.774,34.230,-74.513,171.105,31.127,155.832
C07992=1054.768,33.981,-74.497,171.103,31.125,155.832
C07993=1054.762,33.732,-74.481,171.102,31.123,155.831
C07994=1054.756,33.482,-74.464,171.100,31.120,155.831
C07995=1054.749,33.233,-74.448,171.098,31.118,155.831
C07996=1054.743,32.983,-74.432,171.097,31.116,155.830
C07997=1054.737,32.734,-74.416,171.096,31.114,155.830
C07998=1054.731,32.485,-74.400,171.094,31.111,155.830
C07999=1054.725,32.235,-74.383,171.092,31.109,155.829
C08000=1054.719,31.986,-74.368,171.091,31.107,155.829
C08001=1054.713,31.736,-74.352,171.089,31.105,155.829
C08002=1054.707,31.487,-74.336,171.087,31.103,155.828
C08003=1054.700,31.237,-74.319,171.085,31.100,155.828
C08004=1054.694,30.988,-74.303,171.085,31.098,155.828
C08005=1054.688,30.738,-74.287,171.083,31.096,155.827
C08006=1054.682,30.489,-74.271,171.081,31.094,155.827
C08007=1054.676,30.240,-74.255,171.080,31.092,155.827
C08008=1054.669,29.954,-74.237,171.078,31.089,155.826
C08009=1054.662,29.669,-74.218,171.076,31.086,155.826
C08010=1054.655,29.383,-74.200,171.075,31.084,155.826
C08011=1054.648,29.097,-74.181,171.073,31.081,155.825
C08012=1054.641,28.848,-74.166,171.071,31.079,155.825
C08013=1054.635,28.599,-74.149,171.069,31.077,155.825
C08014=1054.629,28.349,-74.133,171.068,31.075,155.824
C08015=1054.623,28.100,-74.118,171.066,31.073,155.824
C08016=1054.617,27.850,-74.102,171.064,31.070,155.824
C08017=1054.611,27.601,-74.086,171.063,31.068,155.823
C08018=1054.604,27.352,-74.070,171.062,31.066,155.823
C08019=1054.599,27.102,-74.054,171.060,31.064,155.823
C08020=1054.593,26.853,-74.038,171.058,31.062,155.822
C08021=1054.586,26.603,-74.023,171.056,31.059,155.822
C08022=1054.580,26.354,-74.006,171.055,31.057,155.822
C08023=1054.574,26.105,-73.991,171.054,31.055,155.821
C08024=1054.568,25.855,-73.975,171.052,31.053,155.821
C08025=1054.562,25.606,-73.959,171.050,31.051,155.821
C08026=1054.555,25.357,-73.943,171.049,31.049,155.821
C08027=1054.549,25.106,-73.927,171.047,31.046,155.820
C08028=1054.542,24.857,-73.912,171.045,31.044,155.820
C08029=1054.536,24.608,-73.895,171.043,31.042,155.820
C08030=1054.530,24.358,-73.880,171.043,31.040,155.819
C08031=1054.524,24.109,-73.864,171.041,31.038,155.819
C08032=1054.517,23.860,-73.849,171.039,31.035,155.819
C08033=1054.512,23.610,-73.833,171.037,31.033,155.818
C08034=1054.506,23.360,-73.817,171.036,31.031,155.818
C08035=1054.499,23.111,-73.801,171.034,31.029,155.818
C08036=1054.493,22.861,-73.786,171.033,31.027,155.817
C08037=1054.487,22.612,-73.770,171.032,31.025,155.817
C08038=1054.481,22.363,-73.754,171.030,31.022,155.817
C08039=1054.474,22.113,-73.739,171.028,31.020,155.816
C08040=1054.469,21.865,-73.723,171.026,31.018,155.816
C08041=1054.463,21.615,-73.708,171.025,31.016,155.816
C08042=1054.457,21.366,-73.692,171.023,31.014,155.815
C08043=1054.450,21.117,-73.676,171.022,31.011,155.815
C08044=1054.444,20.867,-73.660,171.020,31.009,155.815
C08045=1054.438,20.618,-73.645,171.019,31.007,155.815
C08046=1054.432,20.368,-73.629,171.017,31.005,155.814
C08047=1054.426,20.118,-73.613,171.015,31.002,155.814
C08048=1054.420,19.869,-73.598,171.013,31.000,155.814
C08049=1054.413,19.620,-73.582,171.013,30.998,155.813
C08050=1054.407,19.370,-73.567,171.011,30.996,155.813
C08051=1054.401,19.121,-73.551,171.009,30.994,155.813
C08052=1054.395,18.871,-73.536,171.007,30.992,155.812
C08053=1054.388,18.622,-73.520,171.006,30.990,155.812
C08054=1054.382,18.372,-73.505,171.004,30.987,155.812
C08055=1054.376,18.123,-73.489,171.002,30.985,155.811
C08056=1054.370,17.873,-73.474,171.001,30.983,155.811
C08057=1054.364,17.624,-73.457,170.999,30.981,155.811
C08058=1054.357,17.374,-73.443,170.998,30.979,155.811
C08059=1054.352,17.125,-73.428,170.996,30.977,155.810
C08060=1054.346,16.876,-73.412,170.994,30.975,155.810
C08061=1054.339,16.626,-73.397,170.992,30.973,155.810
C08062=1054.333,16.377,-73.380,170.991,30.971,155.809
C08063=1054.327,16.127,-73.366,170.990,30.968,155.809
C08064=1054.320,15.878,-73.350,170.988,30.966,155.809
C08065=1054.315,15.628,-73.334,170.986,30.964,155.808
C08066=1054.308,15.378,-73.319,170.985,30.962,155.808
C08067=1054.301,15.129,-73.304,170.983,30.960,155.808
C08068=1054.296,14.880,-73.289,170.981,30.958,155.808
C08069=1054.290,14.630,-73.274,170.980,30.955,155.807
C08070=1054.284,14.381,-73.257,170.979,30.953,155.807
C08071=1054.278,14.131,-73.242,170.977,30.951,155.807
C08072=1054.271,13.847,-73.225,170.975,30.949,155.806
C08073=1054.263,13.563,-73.208,170.973,30.946,155.806
C08074=1054.256,13.279,-73.190,170.971,30.944,155.806
C08075=1054.249,12.994,-73.173,170.970,30.942,155.805
C08076=1054.243,12.745,-73.158,170.968,30.939,155.805
C08077=1054.236,12.496,-73.142,170.966,30.937,155.805
C08078=1054.229,12.246,-73.127,170.964,30.935,155.804
C08079=1054.224,11.996,-73.112,170.963,30.933,155.804
C08080=1054.217,11.746,-73.097,170.961,30.931,155.804
C08081=1054.211,11.498,-73.082,170.960,30.929,155.804
C08082=1054.205,11.248,-73.067,170.958,30.927,155.803
C08083=1054.199,10.999,-73.052,170.956,30.925,155.803
C08084=1054.192,10.749,-73.037,170.955,30.923,155.803
C08085=1054.186,10.499,-73.022,170.953,30.921,155.802
C08086=1054.179,10.250,-73.006,170.951,30.919,155.802
C08087=1054.173,10.000,-72.991,170.949,30.916,155.802
C08088=1054.168,9.751,-72.976,170.948,30.915,155.802
C08089=1054.161,9.502,-72.961,170.947,30.913,155.801
C08090=1054.155,9.252,-72.946,170.945,30.911,155.801
C08091=1054.148,9.003,-72.931,170.943,30.909,155.801
C08092=1054.142,8.753,-72.916,170.941,30.907,155.801
C08093=1054.135,8.504,-72.901,170.940,30.905,155.800
C08094=1054.130,8.255,-72.886,170.939,30.902,155.800
C08095=1054.124,8.005,-72.871,170.937,30.900,155.800
C08096=1054.118,7.755,-72.856,170.935,30.898,155.799
C08097=1054.111,7.505,-72.841,170.933,30.896,155.799
C08098=1054.105,7.256,-72.826,170.932,30.894,155.799
C08099=1054.099,7.007,-72.810,170.930,30.892,155.799
C08100=1054.092,6.758,-72.795,170.928,30.890,155.798
C08101=1054.086,6.508,-72.781,170.927,30.888,155.798
C08102=1054.080,6.258,-72.766,170.925,30.886,155.798
C08103=1054.074,6.010,-72.751,170.924,30.884,155.797
C08104=1054.067,5.760,-72.736,170.922,30.882,155.797
C08105=1054.062,5.510,-72.721,170.920,30.879,155.797
C08106=1054.055,5.260,-72.706,170.918,30.877,155.797
C08107=1054.050,5.011,-72.691,170.917,30.875,155.796
C08108=1054.043,4.762,-72.676,170.916,30.873,155.796
C08109=1054.037,4.512,-72.661,170.914,30.871,155.796
C08110=1054.031,4.262,-72.646,170.912,30.869,155.795
C08111=1054.025,4.013,-72.632,170.910,30.867,155.795
C08112=1054.018,3.764,-72.617,170.908,30.865,155.795
C08113=1054.012,3.514,-72.602,170.908,30.863,155.794
C08114=1054.006,3.264,-72.587,170.906,30.861,155.794
C08115=1054.000,3.015,-72.572,170.904,30.858,155.794
C08116=1053.993,2.766,-72.557,170.902,30.856,155.794
C08117=1053.987,2.516,-72.542,170.900,30.855,155.793
C08118=1053.982,2.267,-72.527,170.899,30.853,155.793
C08119=1053.976,2.017,-72.512,170.897,30.851,155.793
C08120=1053.969,1.768,-72.497,170.896,30.849,155.793
C08121=1053.963,1.519,-72.483,170.894,30.846,155.792
C08122=1053.957,1.269,-72.468,170.892,30.844,155.792
C08123=1053.951,1.019,-72.453,170.891,30.842,155.792
C08124=1053.945,0.770,-72.438,170.889,30.840,155.791
C08125=1053.939,0.521,-72.423,170.887,30.838,155.791
C08126=1053.932,0.270,-72.409,170.886,30.836,155.791
C08127=1053.927,0.021,-72.394,170.884,30.834,155.791
C08128=1053.920,-0.228,-72.379,170.883,30.832,155.790
C08129=1053.914,-0.478,-72.365,170.881,30.830,155.790
C08130=1053.908,-0.727,-72.350,170.879,30.827,155.790
C08131=1053.902,-0.977,-72.335,170.877,30.825,155.789
C08132=1053.895,-1.226,-72.320,170.876,30.823,155.789
C08133=1053.890,-1.475,-72.305,170.874,30.821,155.789
C08134=1053.883,-1.725,-72.291,170.873,30.819,155.789
C08135=1053.878,-1.974,-72.277,170.871,30.817,155.788
C08136=1053.870,-2.257,-72.260,170.869,30.815,155.788
C08137=1053.864,-2.539,-72.243,170.867,30.813,155.788
C08138=1053.857,-2.821,-72.226,170.866,30.810,155.787
C08139=1053.850,-3.104,-72.210,170.864,30.808,155.787
C08140=1053.844,-3.354,-72.195,170.862,30.806,155.787
C08141=1053.838,-3.603,-72.181,170.860,30.804,155.787
C08142=1053.832,-3.853,-72.166,170.858,30.802,155.786
C08143=1053.825,-4.102,-72.152,170.856,30.800,155.786
C08144=1053.819,-4.351,-72.138,170.855,30.798,155.786
C08145=1053.813,-4.601,-72.123,170.854,30.796,155.785
C08146=1053.806,-4.850,-72.108,170.852,30.794,155.785
C08147=1053.800,-5.100,-72.094,170.850,30.792,155.785
C08148=1053.794,-5.350,-72.079,170.848,30.790,155.785
C08149=1053.788,-5.599,-72.065,170.846,30.788,155.784
C08150=1053.781,-5.849,-72.051,170.845,30.786,155.784
C08151=1053.775,-6.098,-72.036,170.844,30.784,155.784
C08152=1053.769,-6.347,-72.022,170.842,30.782,155.784
C08153=1053.763,-6.597,-72.007,170.840,30.780,155.783
C08154=1053.756,-6.847,-71.993,170.838,30.778,155.783
C08155=1053.750,-7.096,-71.978,170.836,30.776,155.783
C08156=1053.744,-7.346,-71.964,170.835,30.774,155.783
C08157=1053.737,-7.595,-71.950,170.833,30.772,155.782
C08158=1053.731,-7.845,-71.936,170.832,30.770,155.782
C08159=1053.726,-8.094,-71.921,170.830,30.769,155.782
C08160=1053.719,-8.344,-71.907,170.828,30.766,155.782
C08161=1053.712,-8.594,-71.893,170.826,30.764,155.781
C08162=1053.707,-8.843,-71.878,170.824,30.762,155.781
C08163=1053.700,-9.093,-71.864,170.823,30.761,155.781
C08164=1053.694,-9.341,-71.850,170.821,30.759,155.781
C08165=1053.688,-9.592,-71.836,170.820,30.757,155.780
C08166=1053.682,-9.841,-71.821,170.818,30.754,155.780
C08167=1053.675,-10.090,-71.807,170.816,30.753,155.780
C08168=1053.670,-10.340,-71.793,170.814,30.751,155.780
C08169=1053.663,-10.589,-71.778,170.813,30.749,155.779
C08170=1053.658,-10.839,-71.764,170.811,30.746,155.779
C08171=1053.651,-11.088,-71.750,170.809,30.745,155.779
C08172=1053.645,-11.338,-71.736,170.808,30.743,155.779
C08173=1053.639,-11.587,-71.721,170.806,30.741,155.778
C08174=1053.632,-11.837,-71.708,170.804,30.739,155.778
C08175=1053.626,-12.086,-71.693,170.803,30.737,155.778
C08176=1053.621,-12.336,-71.679,170.801,30.735,155.778
C08177=1053.613,-12.585,-71.665,170.799,30.733,155.777
C08178=1053.608,-12.835,-71.651,170.797,30.731,155.777
C08179=1053.602,-13.085,-71.637,170.796,30.729,155.777
C08180=1053.595,-13.334,-71.623,170.794,30.727,155.777
C08181=1053.589,-13.584,-71.608,170.793,30.725,155.776
C08182=1053.584,-13.833,-71.594,170.791,30.724,155.776
C08183=1053.577,-14.083,-71.580,170.789,30.721,155.776
C08184=1053.571,-14.332,-71.566,170.787,30.719,155.776
C08185=1053.564,-14.582,-71.552,170.785,30.717,155.775
C08186=1053.559,-14.831,-71.538,170.784,30.716,155.775
C08187=1053.552,-15.081,-71.523,170.782,30.714,155.775
C08188=1053.546,-15.330,-71.510,170.781,30.711,155.775
C08189=1053.540,-15.581,-71.496,170.779,30.710,155.774
C08190=1053.533,-15.829,-71.482,170.777,30.708,155.774
C08191=1053.528,-16.079,-71.468,170.775,30.706,155.774
C08192=1053.521,-16.329,-71.454,170.773,30.704,155.774
C08193=1053.515,-16.577,-71.440,170.771,30.702,155.773
C08194=1053.509,-16.828,-71.426,170.770,30.700,155.773
C08195=1053.502,-17.077,-71.413,170.769,30.698,155.773
C08196=1053.496,-17.327,-71.398,170.767,30.697,155.773
C08197=1053.490,-17.576,-71.384,170.765,30.695,155.772
C08198=1053.484,-17.826,-71.370,170.763,30.693,155.772
C08199=1053.477,-18.075,-71.357,170.761,30.691,155.772
C08200=1053.472,-18.301,-71.343,170.760,30.689,155.772
C08201=1053.466,-18.526,-71.331,170.759,30.687,155.772
C08202=1053.460,-18.752,-71.319,170.757,30.686,155.771
C08203=1053.455,-18.977,-71.307,170.755,30.684,155.771
C08204=1053.449,-19.204,-71.294,170.753,30.682,155.771
C08205=1053.443,-19.429,-71.281,170.752,30.681,155.771
C08206=1053.438,-19.655,-71.269,170.750,30.679,155.771
C08207=1053.432,-19.881,-71.257,170.749,30.677,155.770
C08208=1053.426,-20.130,-71.242,170.747,30.676,155.770
C08209=1053.420,-20.379,-71.229,170.745,30.674,155.770
C08210=1053.413,-20.629,-71.215,170.744,30.672,155.770
C08211=1053.408,-20.878,-71.201,170.742,30.670,155.769
C08212=1053.401,-21.128,-71.188,170.740,30.668,155.769
C08213=1053.395,-21.378,-71.174,170.738,30.666,155.769
C08214=1053.389,-21.627,-71.160,170.737,30.665,155.769
C08215=1053.382,-21.877,-71.146,170.735,30.663,155.768
C08216=1053.377,-22.126,-71.132,170.733,30.661,155.768
C08217=1053.370,-22.375,-71.119,170.731,30.659,155.768
C08218=1053.364,-22.626,-71.105,170.729,30.657,155.768
C08219=1053.358,-22.875,-71.092,170.727,30.655,155.768
C08220=1053.352,-23.124,-71.078,170.727,30.653,155.767
C08221=1053.346,-23.375,-71.064,170.725,30.652,155.767
C08222=1053.339,-23.623,-71.050,170.723,30.650,155.767
C08223=1053.333,-23.872,-71.037,170.721,30.648,155.767
C08224=1053.327,-24.123,-71.023,170.719,30.646,155.766
C08225=1053.321,-24.372,-71.009,170.717,30.644,155.766
C08226=1053.315,-24.622,-70.995,170.716,30.642,155.766
C08227=1053.308,-24.872,-70.982,170.714,30.641,155.766
C08228=1053.302,-25.121,-70.968,170.712,30.638,155.766
C08229=1053.297,-25.370,-70.955,170.710,30.637,155.765
C08230=1053.290,-25.620,-70.941,170.708,30.635,155.765
C08231=1053.284,-25.870,-70.928,170.707,30.633,155.765
C08232=1053.278,-26.119,-70.914,170.705,30.631,155.765
C08233=1053.272,-26.368,-70.901,170.704,30.630,155.764
C08234=1053.265,-26.618,-70.887,170.702,30.628,155.764
C08235=1053.260,-26.868,-70.873,170.700,30.625,155.764
C08236=1053.253,-27.117,-70.860,170.698,30.624,155.764
C08237=1053.247,-27.367,-70.846,170.696,30.622,155.764
C08238=1053.240,-27.616,-70.833,170.694,30.620,155.763
C08239=1053.234,-27.866,-70.820,170.693,30.619,155.763
C08240=1053.227,-28.116,-70.806,170.691,30.617,155.763
C08241=1053.222,-28.365,-70.792,170.689,30.615,155.763
C08242=1053.216,-28.615,-70.779,170.687,30.613,155.763
C08243=1053.210,-28.864,-70.766,170.685,30.612,155.762
C08244=1053.203,-29.114,-70.753,170.683,30.610,155.762
C08245=1053.197,-29.364,-70.739,170.682,30.608,155.762
C08246=1053.191,-29.613,-70.726,170.681,30.606,155.762
C08247=1053.184,-29.862,-70.713,170.679,30.605,155.761
C08248=1053.178,-30.112,-70.699,170.677,30.603,155.761
C08249=1053.171,-30.361,-70.686,170.675,30.601,155.761
C08250=1053.166,-30.611,-70.672,170.673,30.599,155.761
C08251=1053.159,-30.861,-70.658,170.671,30.598,155.761
C08252=1053.153,-31.111,-70.646,170.670,30.596,155.760
C08253=1053.147,-31.360,-70.633,170.668,30.594,155.760
C08254=1053.141,-31.609,-70.619,170.666,30.593,155.760
C08255=1053.135,-31.859,-70.606,170.664,30.590,155.760
C08256=1053.126,-32.188,-70.588,170.661,30.588,155.760
C08257=1053.118,-32.517,-70.572,170.660,30.586,155.759
C08258=1053.110,-32.845,-70.554,170.657,30.584,155.759
C08259=1053.101,-33.173,-70.537,170.655,30.581,155.759
C08260=1053.096,-33.423,-70.523,170.653,30.580,155.759
C08261=1053.089,-33.673,-70.509,170.651,30.578,155.758
C08262=1053.083,-33.923,-70.497,170.649,30.576,155.758
C08263=1053.077,-34.172,-70.483,170.648,30.575,155.758
C08264=1053.070,-34.452,-70.468,170.646,30.573,155.758
C08265=1053.063,-34.732,-70.454,170.644,30.571,155.758
C08266=1053.056,-35.012,-70.439,170.641,30.569,155.757
C08267=1053.049,-35.292,-70.425,170.639,30.566,155.757
C08268=1053.043,-35.542,-70.411,170.637,30.565,155.757
C08269=1053.037,-35.791,-70.398,170.636,30.563,155.757
C08270=1053.030,-36.041,-70.385,170.634,30.562,155.757
C08271=1053.024,-36.290,-70.372,170.632,30.560,155.756
C08272=1053.018,-36.539,-70.359,170.630,30.558,155.756
C08273=1053.012,-36.789,-70.346,170.628,30.557,155.756
C08274=1053.006,-37.038,-70.333,170.626,30.554,155.756
C08275=1053.001,-37.289,-70.320,170.625,30.553,155.756
C08276=1052.994,-37.539,-70.306,170.624,30.552,155.755
C08277=1052.988,-37.788,-70.293,170.622,30.549,155.755
C08278=1052.982,-38.038,-70.280,170.620,30.548,155.755
C08279=1052.976,-38.287,-70.267,170.618,30.546,155.755
C08280=1052.969,-38.536,-70.254,170.616,30.545,155.755
C08281=1052.963,-38.786,-70.241,170.614,30.543,155.754
C08282=1052.956,-39.035,-70.228,170.613,30.541,155.754
C08283=1052.951,-39.285,-70.216,170.611,30.539,155.754
C08284=1052.944,-39.535,-70.202,170.609,30.538,155.754
C08285=1052.938,-39.785,-70.190,170.607,30.536,155.754
C08286=1052.932,-40.034,-70.176,170.605,30.535,155.754
C08287=1052.926,-40.284,-70.164,170.603,30.533,155.753
C08288=1052.919,-40.533,-70.151,170.601,30.532,155.753
C08289=1052.913,-40.783,-70.139,170.600,30.530,155.753
C08290=1052.907,-41.032,-70.125,170.598,30.528,155.753
C08291=1052.901,-41.282,-70.113,170.596,30.526,155.753
C08292=1052.895,-41.531,-70.099,170.594,30.525,155.752
C08293=1052.888,-41.782,-70.086,170.592,30.523,155.752
C08294=1052.881,-42.031,-70.074,170.590,30.522,155.752
C08295=1052.875,-42.281,-70.061,170.589,30.520,155.752
C08296=1052.869,-42.530,-70.048,170.587,30.519,155.752
C08297=1052.863,-42.780,-70.035,170.585,30.516,155.752
C08298=1052.857,-43.029,-70.022,170.583,30.515,155.751
C08299=1052.850,-43.279,-70.010,170.581,30.513,155.751
C08300=1052.844,-43.528,-69.998,170.579,30.512,155.751
C08301=1052.838,-43.778,-69.984,170.577,30.510,155.751
C08302=1052.832,-44.028,-69.972,170.576,30.509,155.751
C08303=1052.826,-44.277,-69.959,170.574,30.507,155.751
C08304=1052.819,-44.526,-69.947,170.572,30.506,155.750
C08305=1052.813,-44.776,-69.934,170.570,30.504,155.750
C08306=1052.807,-45.026,-69.921,170.568,30.503,155.750
C08307=1052.801,-45.275,-69.908,170.566,30.501,155.750
C08308=1052.794,-45.524,-69.896,170.565,30.499,155.750
C08309=1052.788,-45.774,-69.883,170.563,30.497,155.749
C08310=1052.782,-46.024,-69.870,170.561,30.496,155.749
C08311=1052.776,-46.273,-69.857,170.559,30.494,155.749
C08312=1052.770,-46.523,-69.845,170.557,30.493,155.749
C08313=1052.764,-46.773,-69.833,170.555,30.491,155.749
C08314=1052.757,-47.022,-69.819,170.553,30.489,155.749
C08315=1052.752,-47.272,-69.807,170.552,30.488,155.749
C08316=1052.746,-47.522,-69.794,170.550,30.486,155.748
C08317=1052.739,-47.772,-69.782,170.548,30.485,155.748
C08318=1052.733,-48.021,-69.769,170.546,30.483,155.748
C08319=1052.727,-48.271,-69.757,170.544,30.482,155.748
C08320=1052.721,-48.521,-69.744,170.542,30.480,155.748
C08321=1052.714,-48.769,-69.731,170.541,30.479,155.748
C08322=1052.708,-49.019,-69.719,170.539,30.477,155.747
C08323=1052.702,-49.269,-69.706,170.537,30.475,155.747
C08324=1052.696,-49.519,-69.694,170.535,30.474,155.747
C08325=1052.690,-49.769,-69.682,170.533,30.472,155.747
C08326=1052.683,-50.018,-69.668,170.531,30.471,155.747
C08327=1052.678,-50.268,-69.656,170.529,30.469,155.747
C08328=1052.671,-50.548,-69.643,170.527,30.468,155.746
C08329=1052.664,-50.828,-69.629,170.525,30.466,155.746
C08330=1052.656,-51.109,-69.615,170.523,30.464,155.746
C08331=1052.649,-51.389,-69.600,170.521,30.462,155.746
C08332=1052.643,-51.638,-69.588,170.519,30.461,155.746
C08333=1052.637,-51.888,-69.576,170.516,30.460,155.746
C08334=1052.630,-52.138,-69.564,170.515,30.458,155.746
C08335=1052.624,-52.388,-69.551,170.513,30.456,155.745
C08336=1052.618,-52.637,-69.539,170.511,30.456,155.745
C08337=1052.611,-52.887,-69.527,170.509,30.454,155.745
C08338=1052.605,-53.137,-69.515,170.507,30.452,155.745
C08339=1052.598,-53.386,-69.503,170.505,30.451,155.745
C08340=1052.592,-53.636,-69.490,170.503,30.449,155.745
C08341=1052.586,-53.886,-69.478,170.502,30.448,155.745
C08342=1052.580,-54.135,-69.465,170.500,30.447,155.744
C08343=1052.573,-54.385,-69.453,170.498,30.445,155.744
C08344=1052.566,-54.634,-69.441,170.496,30.444,155.744
C08345=1052.560,-54.884,-69.429,170.494,30.443,155.744
C08346=1052.554,-55.133,-69.417,170.492,30.441,155.744
C08347=1052.548,-55.383,-69.405,170.490,30.440,155.744
C08348=1052.542,-55.632,-69.393,170.489,30.438,155.744
C08349=1052.535,-55.882,-69.381,170.487,30.437,155.744
C08350=1052.529,-56.132,-69.368,170.485,30.436,155.743
C08351=1052.523,-56.381,-69.356,170.483,30.434,155.743
C08352=1052.516,-56.631,-69.344,170.481,30.432,155.743
C08353=1052.510,-56.881,-69.332,170.479,30.431,155.743
C08354=1052.504,-57.131,-69.320,170.476,30.430,155.743
C08355=1052.498,-57.380,-69.308,170.475,30.428,155.743
C08356=1052.492,-57.630,-69.296,170.473,30.427,155.743
C08357=1052.485,-57.879,-69.284,170.471,30.426,155.743
C08358=1052.479,-58.129,-69.272,170.469,30.424,155.742
C08359=1052.473,-58.379,-69.260,170.467,30.423,155.742
C08360=1052.466,-58.628,-69.248,170.465,30.421,155.742
C08361=1052.460,-58.878,-69.235,170.463,30.420,155.742
C08362=1052.454,-59.127,-69.224,170.462,30.418,155.742
C08363=1052.448,-59.377,-69.211,170.460,30.417,155.742
C08364=1052.441,-59.627,-69.199,170.458,30.416,155.742
C08365=1052.435,-59.877,-69.188,170.456,30.414,155.742
C08366=1052.429,-60.127,-69.175,170.454,30.413,155.741
C08367=1052.423,-60.376,-69.164,170.452,30.412,155.741
C08368=1052.416,-60.625,-69.152,170.450,30.410,155.741
C08369=1052.411,-60.875,-69.139,170.448,30.409,155.741
C08370=1052.404,-61.125,-69.127,170.447,30.408,155.741
C08371=1052.397,-61.374,-69.115,170.444,30.406,155.741
C08372=1052.392,-61.624,-69.104,170.442,30.405,155.741
C08373=1052.386,-61.873,-69.092,170.440,30.404,155.741
C08374=1052.379,-62.123,-69.080,170.438,30.402,155.740
C08375=1052.373,-62.373,-69.067,170.436,30.400,155.740
C08376=1052.367,-62.622,-69.056,170.434,30.400,155.740
C08377=1052.361,-62.872,-69.045,170.433,30.398,155.740
C08378=1052.355,-63.122,-69.032,170.431,30.396,155.740
C08379=1052.348,-63.371,-69.020,170.429,30.395,155.740
C08380=1052.342,-63.620,-69.008,170.427,30.394,155.740
C08381=1052.336,-63.871,-68.997,170.425,30.392,155.740
C08382=1052.330,-64.120,-68.985,170.423,30.391,155.740
C08383=1052.323,-64.370,-68.973,170.421,30.390,155.739
C08384=1052.317,-64.619,-68.962,170.420,30.388,155.739
C08385=1052.312,-64.869,-68.949,170.417,30.387,155.739
C08386=1052.305,-65.119,-68.937,170.415,30.386,155.739
C08387=1052.299,-65.368,-68.926,170.413,30.385,155.739
C08388=1052.293,-65.618,-68.914,170.411,30.383,155.739
C08389=1052.287,-65.868,-68.902,170.409,30.381,155.739
C08390=1052.281,-66.117,-68.890,170.407,30.381,155.739
C08391=1052.275,-66.367,-68.878,170.406,30.379,155.738
C08392=1052.267,-66.649,-68.865,170.404,30.377,155.738
C08393=1052.261,-66.930,-68.852,170.401,30.376,155.738
C08394=1052.254,-67.212,-68.838,170.399,30.375,155.738
C08395=1052.246,-67.493,-68.826,170.397,30.373,155.738
C08396=1052.241,-67.744,-68.814,170.395,30.372,155.738
C08397=1052.235,-67.993,-68.802,170.393,30.370,155.738
C08398=1052.228,-68.243,-68.791,170.391,30.369,155.738
C08399=1052.223,-68.493,-68.778,170.389,30.368,155.738
C08400=1052.217,-68.742,-68.767,170.387,30.366,155.737
C08401=1052.210,-68.992,-68.755,170.385,30.365,155.737
C08402=1052.204,-69.241,-68.744,170.383,30.364,155.737
C08403=1052.199,-69.491,-68.732,170.381,30.362,155.737
C08404=1052.192,-69.741,-68.720,170.379,30.361,155.737
C08405=1052.186,-69.990,-68.709,170.378,30.360,155.737
C08406=1052.180,-70.240,-68.697,170.376,30.359,155.737
C08407=1052.174,-70.490,-68.685,170.374,30.357,155.737
C08408=1052.168,-70.739,-68.674,170.372,30.356,155.737
C08409=1052.161,-70.989,-68.662,170.369,30.355,155.737
C08410=1052.155,-71.238,-68.651,170.367,30.354,155.737
C08411=1052.150,-71.488,-68.638,170.365,30.352,155.736
C08412=1052.144,-71.738,-68.628,170.364,30.351,155.736
C08413=1052.137,-71.987,-68.616,170.362,30.350,155.736
C08414=1052.131,-72.237,-68.604,170.360,30.349,155.736
C08415=1052.125,-72.487,-68.593,170.358,30.347,155.736
C08416=1052.119,-72.737,-68.581,170.356,30.346,155.736
C08417=1052.113,-72.986,-68.570,170.354,30.344,155.736
C08418=1052.107,-73.236,-68.558,170.352,30.344,155.736
C08419=1052.101,-73.485,-68.547,170.350,30.342,155.736
C08420=1052.095,-73.735,-68.535,170.348,30.341,155.736
C08421=1052.089,-73.985,-68.524,170.346,30.339,155.735
C08422=1052.083,-74.235,-68.513,170.344,30.338,155.735
C08423=1052.077,-74.484,-68.501,170.342,30.337,155.735
C08424=1052.071,-74.734,-68.490,170.340,30.336,155.735
C08425=1052.064,-74.984,-68.478,170.338,30.335,155.735
C08426=1052.058,-75.233,-68.467,170.336,30.333,155.735
C08427=1052.052,-75.483,-68.456,170.335,30.332,155.735
C08428=1052.046,-75.732,-68.444,170.333,30.331,155.735
C08429=1052.040,-75.982,-68.433,170.330,30.330,155.735
C08430=1052.034,-76.232,-68.422,170.328,30.329,155.735
C08431=1052.027,-76.481,-68.410,170.326,30.328,155.735
C08432=1052.021,-76.731,-68.399,170.324,30.327,155.735
C08433=1052.015,-76.981,-68.388,170.322,30.325,155.734
C08434=1052.009,-77.231,-68.377,170.320,30.324,155.734
C08435=1052.002,-77.480,-68.366,170.319,30.323,155.734
C08436=1051.996,-77.730,-68.354,170.317,30.322,155.734
C08437=1051.990,-77.980,-68.343,170.314,30.321,155.734
C08438=1051.983,-78.229,-68.331,170.312,30.320,155.734
C08439=1051.978,-78.479,-68.321,170.310,30.319,155.734
C08440=1051.971,-78.729,-68.309,170.308,30.317,155.734
C08441=1051.965,-78.978,-68.298,170.306,30.316,155.734
C08442=1051.960,-79.228,-68.288,170.304,30.315,155.734
C08443=1051.953,-79.477,-68.276,170.303,30.314,155.734
C08444=1051.947,-79.727,-68.265,170.301,30.313,155.734
C08445=1051.941,-79.977,-68.254,170.298,30.312,155.734
C08446=1051.935,-80.226,-68.243,170.296,30.311,155.734
C08447=1051.928,-80.476,-68.232,170.294,30.310,155.734
C08448=1051.922,-80.726,-68.220,170.292,30.309,155.733
C08449=1051.916,-80.975,-68.209,170.290,30.308,155.733
C08450=1051.909,-81.226,-68.198,170.288,30.307,155.733
C08451=1051.903,-81.475,-68.188,170.287,30.306,155.733
C08452=1051.897,-81.725,-68.176,170.284,30.305,155.733
C08453=1051.891,-81.974,-68.166,170.282,30.304,155.733
C08454=1051.884,-82.224,-68.155,170.280,30.303,155.733
C08455=1051.878,-82.474,-68.144,170.278,30.302,155.733
C08456=1051.871,-82.758,-68.131,170.276,30.300,155.733
C08457=1051.864,-83.042,-68.119,170.273,30.299,155.733
C08458=1051.857,-83.326,-68.106,170.271,30.298,155.733
C08459=1051.850,-83.609,-68.094,170.269,30.297,155.733
C08460=1051.843,-83.859,-68.083,170.267,30.296,155.733
C08461=1051.838,-84.109,-68.072,170.265,30.295,155.733
C08462=1051.831,-84.358,-68.062,170.263,30.294,155.733
C08463=1051.825,-84.608,-68.051,170.261,30.293,155.733
C08464=1051.819,-84.858,-68.039,170.259,30.292,155.733
C08465=1051.812,-85.107,-68.029,170.256,30.291,155.733
C08466=1051.806,-85.358,-68.018,170.254,30.290,155.733
C08467=1051.800,-85.607,-68.007,170.253,30.289,155.733
C08468=1051.794,-85.856,-67.996,170.251,30.288,155.733
C08469=1051.787,-86.106,-67.986,170.249,30.287,155.733
C08470=1051.781,-86.356,-67.975,170.247,30.286,155.733
C08471=1051.775,-86.606,-67.963,170.245,30.285,155.733
C08472=1051.769,-86.855,-67.953,170.242,30.284,155.733
C08473=1051.763,-87.105,-67.942,170.240,30.283,155.732
C08474=1051.757,-87.355,-67.931,170.238,30.282,155.732
C08475=1051.750,-87.604,-67.921,170.236,30.281,155.732
C08476=1051.744,-87.854,-67.910,170.235,30.280,155.732
C08477=1051.738,-88.104,-67.899,170.233,30.279,155.732
C08478=1051.731,-88.353,-67.888,170.230,30.278,155.732
C08479=1051.726,-88.602,-67.877,170.228,30.277,155.732
C08480=1051.719,-88.853,-67.866,170.226,30.276,155.732
C08481=1051.713,-89.102,-67.856,170.224,30.275,155.732
C08482=1051.708,-89.352,-67.846,170.222,30.274,155.732
C08483=1051.701,-89.602,-67.835,170.220,30.274,155.732
C08484=1051.695,-89.851,-67.824,170.218,30.272,155.732
C08485=1051.689,-90.101,-67.813,170.216,30.271,155.732
C08486=1051.683,-90.351,-67.802,170.214,30.270,155.732
C08487=1051.676,-90.600,-67.792,170.212,30.270,155.732
C08488=1051.670,-90.850,-67.781,170.210,30.269,155.732
C08489=1051.664,-91.100,-67.771,170.208,30.268,155.732
C08490=1051.658,-91.350,-67.760,170.206,30.267,155.732
C08491=1051.652,-91.599,-67.749,170.203,30.266,155.732
C08492=1051.645,-91.849,-67.739,170.201,30.265,155.732
C08493=1051.639,-92.098,-67.728,170.200,30.264,155.732
C08494=1051.634,-92.349,-67.718,170.198,30.263,155.732
C08495=1051.627,-92.598,-67.707,170.196,30.262,155.732
C08496=1051.621,-92.848,-67.696,170.194,30.261,155.732
C08497=1051.615,-93.097,-67.686,170.191,30.261,155.732
C08498=1051.609,-93.347,-67.675,170.189,30.260,155.732
C08499=1051.603,-93.597,-67.665,170.187,30.259,155.732
C08500=1051.596,-93.847,-67.654,170.185,30.258,155.732
C08501=1051.591,-94.096,-67.643,170.183,30.257,155.732
C08502=1051.584,-94.346,-67.634,170.182,30.256,155.732
C08503=1051.579,-94.595,-67.623,170.179,30.255,155.732
C08504=1051.573,-94.845,-67.612,170.177,30.255,155.732
C08505=1051.566,-95.095,-67.601,170.175,30.254,155.732
C08506=1051.560,-95.345,-67.591,170.173,30.253,155.732
C08507=1051.554,-95.594,-67.581,170.171,30.252,155.732
C08508=1051.548,-95.844,-67.570,170.169,30.251,155.731
C08509=1051.543,-96.094,-67.560,170.166,30.250,155.732
C08510=1051.536,-96.344,-67.549,170.164,30.249,155.732
C08511=1051.530,-96.593,-67.538,170.163,30.248,155.731
C08512=1051.524,-96.843,-67.529,170.161,30.247,155.731
C08513=1051.518,-97.092,-67.518,170.159,30.246,155.731
C08514=1051.513,-97.342,-67.508,170.157,30.246,155.731
C08515=1051.506,-97.592,-67.497,170.154,30.245,155.731
C08516=1051.499,-97.841,-67.487,170.152,30.244,155.731
C08517=1051.494,-98.092,-67.477,170.150,30.244,155.731
C08518=1051.487,-98.341,-67.466,170.148,30.243,155.731
C08519=1051.480,-98.591,-67.456,170.146,30.242,155.731
C08520=1051.474,-98.878,-67.444,170.144,30.241,155.732
C08521=1051.467,-99.164,-67.433,170.142,30.240,155.731
C08522=1051.460,-99.450,-67.421,170.139,30.239,155.731
C08523=1051.453,-99.736,-67.409,170.137,30.239,155.732
C08524=1051.446,-99.985,-67.399,170.135,30.238,155.731
C08525=1051.441,-100.236,-67.389,170.132,30.237,155.731
C08526=1051.434,-100.485,-67.378,170.130,30.236,155.732
C08527=1051.428,-100.734,-67.369,170.128,30.235,155.732
C08528=1051.422,-100.984,-67.358,170.126,30.235,155.732
C08529=1051.416,-101.234,-67.348,170.124,30.234,155.732
C08530=1051.409,-101.484,-67.338,170.122,30.233,155.732
C08531=1051.403,-101.734,-67.327,170.120,30.233,155.732
C08532=1051.397,-101.983,-67.317,170.118,30.232,155.732
C08533=1051.391,-102.233,-67.308,170.116,30.231,155.732
C08534=1051.385,-102.482,-67.297,170.114,30.230,155.732
C08535=1051.379,-102.732,-67.287,170.111,30.230,155.732
C08536=1051.372,-102.981,-67.277,170.109,30.229,155.732
C08537=1051.366,-103.231,-67.267,170.107,30.228,155.732
C08538=1051.360,-103.482,-67.257,170.105,30.227,155.732
C08539=1051.354,-103.731,-67.247,170.103,30.227,155.732
C08540=1051.348,-103.981,-67.237,170.102,30.226,155.732
C08541=1051.342,-104.230,-67.226,170.099,30.226,155.732
C08542=1051.336,-104.480,-67.216,170.097,30.225,155.732
C08543=1051.329,-104.730,-67.207,170.095,30.224,155.732
C08544=1051.324,-104.979,-67.196,170.093,30.223,155.732
C08545=1051.318,-105.229,-67.186,170.091,30.223,155.732
C08546=1051.311,-105.479,-67.177,170.088,30.222,155.732
C08547=1051.305,-105.728,-67.167,170.086,30.222,155.732
C08548=1051.300,-105.978,-67.156,170.084,30.221,155.732
C08549=1051.293,-106.228,-67.147,170.082,30.220,155.732
C08550=1051.286,-106.478,-67.136,170.081,30.219,155.732
C08551=1051.280,-106.728,-67.127,170.078,30.219,155.732
C08552=1051.275,-106.978,-67.117,170.076,30.218,155.732
C08553=1051.268,-107.228,-67.107,170.074,30.217,155.732
C08554=1051.262,-107.477,-67.097,170.072,30.217,155.732
C08555=1051.256,-107.727,-67.087,170.070,30.216,155.732
C08556=1051.250,-107.976,-67.078,170.067,30.216,155.732
C08557=1051.243,-108.226,-67.068,170.065,30.215,155.732
C08558=1051.238,-108.476,-67.057,170.063,30.214,155.732
C08559=1051.232,-108.725,-67.048,170.061,30.214,155.732
C08560=1051.225,-108.975,-67.038,170.059,30.214,155.732
C08561=1051.219,-109.225,-67.028,170.057,30.212,155.732
C08562=1051.213,-109.474,-67.018,170.055,30.212,155.732
C08563=1051.207,-109.724,-67.009,170.053,30.212,155.732
C08564=1051.200,-109.974,-66.999,170.051,30.211,155.733
C08565=1051.194,-110.224,-66.989,170.049,30.210,155.733
C08566=1051.188,-110.473,-66.980,170.046,30.210,155.733
C08567=1051.183,-110.724,-66.970,170.044,30.210,155.733
C08568=1051.176,-110.973,-66.959,170.042,30.209,155.733
C08569=1051.170,-111.223,-66.950,170.040,30.208,155.733
C08570=1051.164,-111.472,-66.940,170.037,30.208,155.733
C08571=1051.158,-111.722,-66.931,170.035,30.207,155.733
C08572=1051.151,-111.972,-66.921,170.033,30.206,155.733
C08573=1051.145,-112.222,-66.912,170.032,30.206,155.733
C08574=1051.139,-112.472,-66.902,170.030,30.206,155.733
C08575=1051.133,-112.721,-66.892,170.027,30.205,155.733
C08576=1051.126,-112.970,-66.882,170.025,30.204,155.733
C08577=1051.120,-113.220,-66.873,170.023,30.204,155.733
C08578=1051.114,-113.470,-66.863,170.021,30.204,155.733
C08579=1051.109,-113.720,-66.853,170.019,30.203,155.733
C08580=1051.103,-113.970,-66.843,170.016,30.202,155.733
C08581=1051.096,-114.220,-66.834,170.014,30.202,155.733
C08582=1051.090,-114.470,-66.824,170.012,30.201,155.733
C08583=1051.084,-114.719,-66.815,170.010,30.201,155.733
C08584=1051.077,-115.004,-66.804,170.007,30.201,155.734
C08585=1051.070,-115.289,-66.793,170.006,30.200,155.734
C08586=1051.062,-115.574,-66.782,170.003,30.200,155.734
C08587=1051.056,-115.859,-66.771,170.001,30.199,155.734
C08588=1051.050,-116.108,-66.762,169.998,30.198,155.734
C08589=1051.044,-116.358,-66.752,169.996,30.198,155.734
C08590=1051.038,-116.608,-66.742,169.994,30.198,155.734
C08591=1051.031,-116.857,-66.733,169.992,30.197,155.734
C08592=1051.025,-117.107,-66.725,169.990,30.197,155.734
C08593=1051.019,-117.357,-66.715,169.987,30.196,155.734
C08594=1051.013,-117.607,-66.705,169.985,30.196,155.734
C08595=1051.007,-117.857,-66.696,169.983,30.196,155.734
C08596=1051.000,-118.107,-66.686,169.981,30.195,155.734
C08597=1050.994,-118.356,-66.677,169.979,30.195,155.735
C08598=1050.989,-118.606,-66.668,169.977,30.194,155.735
C08599=1050.983,-118.855,-66.658,169.975,30.194,155.735
C08600=1050.976,-119.105,-66.648,169.973,30.193,155.735
C08601=1050.970,-119.355,-66.639,169.971,30.193,155.735
C08602=1050.964,-119.605,-66.629,169.968,30.192,155.735
C08603=1050.957,-119.855,-66.621,169.966,30.192,155.735
C08604=1050.951,-120.105,-66.611,169.964,30.192,155.735
C08605=1050.946,-120.354,-66.602,169.962,30.191,155.735
C08606=1050.939,-120.604,-66.593,169.959,30.191,155.735
C08607=1050.933,-120.853,-66.583,169.957,30.190,155.735
C08608=1050.927,-121.103,-66.574,169.955,30.191,155.735
C08609=1050.921,-121.354,-66.565,169.953,30.190,155.735
C08610=1050.915,-121.603,-66.555,169.951,30.190,155.736
C08611=1050.909,-121.852,-66.547,169.949,30.189,155.736
C08612=1050.903,-122.102,-66.537,169.947,30.189,155.736
C08613=1050.896,-122.352,-66.527,169.945,30.189,155.736
C08614=1050.891,-122.602,-66.519,169.943,30.188,155.736
C08615=1050.884,-122.852,-66.509,169.940,30.188,155.736
C08616=1050.879,-123.101,-66.500,169.938,30.188,155.736
C08617=1050.872,-123.351,-66.491,169.936,30.187,155.736
C08618=1050.866,-123.601,-66.482,169.934,30.187,155.736
C08619=1050.860,-123.851,-66.472,169.932,30.187,155.736
C08620=1050.854,-124.101,-66.463,169.929,30.186,155.736
C08621=1050.848,-124.350,-66.454,169.927,30.186,155.736
C08622=1050.842,-124.600,-66.445,169.925,30.186,155.737
C08623=1050.835,-124.850,-66.436,169.923,30.186,155.737
C08624=1050.829,-125.099,-66.426,169.920,30.185,155.737
C08625=1050.823,-125.350,-66.417,169.919,30.185,155.737
C08626=1050.817,-125.599,-66.409,169.917,30.184,155.737
C08627=1050.811,-125.848,-66.399,169.915,30.185,155.737
C08628=1050.805,-126.099,-66.390,169.912,30.184,155.737
C08629=1050.798,-126.348,-66.381,169.910,30.184,155.737
C08630=1050.793,-126.597,-66.372,169.908,30.183,155.737
C08631=1050.787,-126.848,-66.363,169.906,30.184,155.737
C08632=1050.780,-127.097,-66.354,169.903,30.183,155.738
C08633=1050.774,-127.347,-66.345,169.901,30.183,155.738
C08634=1050.768,-127.597,-66.336,169.899,30.183,155.738
C08635=1050.762,-127.847,-66.327,169.897,30.182,155.738
C08636=1050.758,-128.097,-66.318,169.895,30.182,155.738
C08637=1050.754,-128.346,-66.307,169.893,30.181,155.738
C08638=1050.750,-128.596,-66.296,169.892,30.179,155.738
C08639=1050.748,-128.846,-66.285,169.890,30.176,155.737
C08640=1050.747,-129.097,-66.272,169.888,30.174,155.737
C08641=1050.747,-129.348,-66.259,169.886,30.171,155.737
C08642=1050.749,-129.598,-66.246,169.886,30.168,155.736
C08643=1050.751,-129.847,-66.232,169.884,30.163,155.735
C08644=1050.754,-130.099,-66.217,169.883,30.158,155.735
C08645=1050.760,-130.350,-66.201,169.883,30.154,155.734
C08646=1050.764,-130.600,-66.185,169.881,30.148,155.733
C08647=1050.771,-130.850,-66.169,169.881,30.141,155.732
C08648=1050.406,-130.873,-66.393,169.835,30.310,155.764
C08649=1050.400,-130.623,-66.409,169.836,30.316,155.765
C08650=1050.395,-130.373,-66.426,169.836,30.321,155.766
C08651=1050.389,-130.122,-66.441,169.838,30.327,155.767
C08652=1050.386,-129.871,-66.456,169.838,30.331,155.767
C08653=1050.384,-129.621,-66.471,169.839,30.335,155.768
C08654=1050.382,-129.371,-66.484,169.841,30.339,155.769
C08655=1050.382,-129.120,-66.497,169.842,30.342,155.769
C08656=1050.383,-128.870,-66.509,169.843,30.345,155.769
C08657=1050.385,-128.620,-66.521,169.845,30.347,155.770
C08658=1050.388,-128.370,-66.531,169.847,30.349,155.770
C08659=1050.391,-128.120,-66.542,169.849,30.350,155.770
C08660=1050.396,-127.870,-66.552,169.851,30.350,155.770
C08661=1050.403,-127.621,-66.561,169.854,30.351,155.770
C08662=1050.409,-127.370,-66.569,169.856,30.351,155.770
C08663=1050.415,-127.121,-66.579,169.857,30.352,155.770
C08664=1050.421,-126.872,-66.588,169.859,30.352,155.770
C08665=1050.427,-126.621,-66.596,169.862,30.352,155.769
C08666=1050.433,-126.372,-66.606,169.864,30.352,155.769
C08667=1050.439,-126.121,-66.615,169.866,30.353,155.769
C08668=1050.445,-125.872,-66.623,169.868,30.353,155.769
C08669=1050.451,-125.623,-66.633,169.871,30.353,155.769
C08670=1050.457,-125.372,-66.642,169.873,30.353,155.769
C08671=1050.464,-125.123,-66.651,169.875,30.353,155.769
C08672=1050.470,-124.874,-66.660,169.877,30.354,155.769
C08673=1050.476,-124.623,-66.669,169.880,30.354,155.769
C08674=1050.482,-124.373,-66.678,169.882,30.354,155.768
C08675=1050.489,-124.124,-66.687,169.884,30.354,155.768
C08676=1050.495,-123.874,-66.697,169.886,30.355,155.768
C08677=1050.500,-123.624,-66.705,169.889,30.355,155.768
C08678=1050.506,-123.375,-66.715,169.890,30.355,155.768
C08679=1050.513,-123.125,-66.725,169.892,30.356,155.768
C08680=1050.519,-122.875,-66.734,169.894,30.356,155.768
C08681=1050.525,-122.625,-66.742,169.896,30.356,155.768
C08682=1050.531,-122.376,-66.752,169.899,30.357,155.768
C08683=1050.537,-122.126,-66.761,169.901,30.357,155.768
C08684=1050.543,-121.876,-66.771,169.903,30.357,155.768
C08685=1050.549,-121.626,-66.780,169.905,30.357,155.768
C08686=1050.555,-121.376,-66.789,169.908,30.358,155.767
C08687=1050.562,-121.127,-66.798,169.910,30.358,155.767
C08688=1050.568,-120.877,-66.807,169.912,30.359,155.767
C08689=1050.574,-120.628,-66.817,169.914,30.359,155.767
C08690=1050.580,-120.378,-66.826,169.917,30.359,155.767
C08691=1050.586,-120.127,-66.835,169.919,30.360,155.767
C08692=1050.592,-119.878,-66.845,169.921,30.360,155.767
C08693=1050.598,-119.628,-66.854,169.922,30.360,155.767
C08694=1050.604,-119.379,-66.864,169.924,30.361,155.767
C08695=1050.611,-119.129,-66.873,169.927,30.361,155.767
C08696=1050.617,-118.879,-66.882,169.929,30.362,155.767
C08697=1050.623,-118.630,-66.892,169.931,30.362,155.767
C08698=1050.629,-118.380,-66.901,169.933,30.362,155.767
C08699=1050.635,-118.129,-66.910,169.936,30.363,155.766
C08700=1050.641,-117.880,-66.920,169.938,30.363,155.766
C08701=1050.647,-117.630,-66.929,169.940,30.363,155.766
C08702=1050.653,-117.381,-66.939,169.942,30.364,155.766
C08703=1050.659,-117.131,-66.948,169.945,30.365,155.766
C08704=1050.665,-116.881,-66.958,169.947,30.365,155.766
C08705=1050.672,-116.631,-66.967,169.949,30.366,155.766
C08706=1050.678,-116.382,-66.977,169.951,30.366,155.766
C08707=1050.684,-116.132,-66.986,169.952,30.366,155.766
C08708=1050.690,-115.882,-66.996,169.955,30.367,155.766
C08709=1050.697,-115.597,-67.007,169.957,30.367,155.766
C08710=1050.704,-115.312,-67.017,169.960,30.368,155.766
C08711=1050.712,-115.027,-67.028,169.962,30.368,155.766
C08712=1050.718,-114.742,-67.039,169.965,30.369,155.766
C08713=1050.724,-114.492,-67.049,169.967,30.369,155.766
C08714=1050.730,-114.242,-67.058,169.969,30.370,155.765
C08715=1050.737,-113.993,-67.068,169.971,30.370,155.765
C08716=1050.743,-113.743,-67.078,169.974,30.371,155.765
C08717=1050.749,-113.493,-67.088,169.976,30.371,155.765
C08718=1050.755,-113.244,-67.097,169.978,30.372,155.765
C08719=1050.761,-112.994,-67.107,169.979,30.372,155.765
C08720=1050.768,-112.744,-67.116,169.982,30.373,155.765
C08721=1050.774,-112.494,-67.126,169.984,30.373,155.765
C08722=1050.779,-112.245,-67.135,169.986,30.374,155.765
C08723=1050.786,-111.995,-67.145,169.988,30.374,155.765
C08724=1050.792,-111.746,-67.154,169.990,30.375,155.765
C08725=1050.798,-111.496,-67.164,169.993,30.375,155.765
C08726=1050.804,-111.246,-67.175,169.995,30.376,155.765
C08727=1050.810,-110.997,-67.184,169.997,30.376,155.765
C08728=1050.816,-110.747,-67.194,169.999,30.377,155.765
C08729=1050.822,-110.497,-67.203,170.001,30.377,155.765
C08730=1050.828,-110.247,-67.213,170.004,30.378,155.765
C08731=1050.834,-109.997,-67.222,170.005,30.379,155.765
C08732=1050.841,-109.748,-67.233,170.007,30.379,155.765
C08733=1050.847,-109.498,-67.242,170.009,30.380,155.765
C08734=1050.853,-109.249,-67.252,170.012,30.380,155.765
C08735=1050.859,-108.998,-67.262,170.014,30.381,155.764
C08736=1050.866,-108.748,-67.272,170.016,30.381,155.764
C08737=1050.872,-108.499,-67.282,170.018,30.382,155.764
C08738=1050.878,-108.249,-67.292,170.020,30.382,155.764
C08739=1050.884,-107.999,-67.301,170.023,30.383,155.764
C08740=1050.891,-107.749,-67.311,170.025,30.384,155.764
C08741=1050.897,-107.500,-67.321,170.027,30.384,155.764
C08742=1050.903,-107.250,-67.331,170.029,30.384,155.764
C08743=1050.909,-107.000,-67.341,170.030,30.385,155.764
C08744=1050.915,-106.750,-67.351,170.033,30.386,155.764
C08745=1050.921,-106.501,-67.361,170.035,30.387,155.764
C08746=1050.927,-106.252,-67.370,170.037,30.387,155.764
C08747=1050.933,-106.001,-67.381,170.039,30.388,155.764
C08748=1050.939,-105.752,-67.391,170.041,30.388,155.764
C08749=1050.946,-105.502,-67.400,170.044,30.389,155.764
C08750=1050.952,-105.253,-67.410,170.046,30.390,155.764
C08751=1050.957,-105.003,-67.421,170.048,30.390,155.764
C08752=1050.964,-104.753,-67.430,170.050,30.391,155.764
C08753=1050.970,-104.503,-67.440,170.052,30.392,155.764
C08754=1050.976,-104.253,-67.451,170.054,30.393,155.764
C08755=1050.982,-104.004,-67.461,170.056,30.393,155.764
C08756=1050.989,-103.754,-67.471,170.058,30.394,155.764
C08757=1050.995,-103.505,-67.481,170.060,30.394,155.764
C08758=1051.000,-103.254,-67.491,170.062,30.395,155.764
C08759=1051.007,-103.005,-67.501,170.065,30.396,155.764
C08760=1051.013,-102.755,-67.511,170.067,30.397,155.764
C08761=1051.019,-102.506,-67.521,170.069,30.397,155.764
C08762=1051.026,-102.255,-67.531,170.071,30.398,155.764
C08763=1051.032,-102.006,-67.542,170.073,30.399,155.764
C08764=1051.037,-101.756,-67.552,170.075,30.399,155.764
C08765=1051.044,-101.506,-67.561,170.077,30.400,155.764
C08766=1051.050,-101.257,-67.572,170.079,30.401,155.764
C08767=1051.056,-101.007,-67.582,170.081,30.402,155.764
C08768=1051.062,-100.758,-67.592,170.083,30.402,155.764
C08769=1051.069,-100.507,-67.602,170.086,30.403,155.764
C08770=1051.074,-100.258,-67.613,170.088,30.404,155.764
C08771=1051.081,-100.008,-67.623,170.090,30.404,155.764
C08772=1051.087,-99.759,-67.633,170.092,30.405,155.764
C08773=1051.093,-99.473,-67.645,170.095,30.406,155.764
C08774=1051.101,-99.186,-67.657,170.097,30.407,155.764
C08775=1051.108,-98.900,-67.669,170.099,30.408,155.764
C08776=1051.115,-98.614,-67.680,170.101,30.408,155.764
C08777=1051.121,-98.364,-67.690,170.103,30.409,155.764
C08778=1051.128,-98.114,-67.701,170.106,30.410,155.764
C08779=1051.134,-97.865,-67.711,170.108,30.411,155.764
C08780=1051.140,-97.615,-67.721,170.110,30.412,155.764
C08781=1051.146,-97.366,-67.732,170.112,30.413,155.764
C08782=1051.152,-97.116,-67.741,170.114,30.413,155.764
C08783=1051.158,-96.866,-67.752,170.116,30.414,155.764
C08784=1051.164,-96.616,-67.763,170.118,30.415,155.764
C08785=1051.170,-96.366,-67.773,170.120,30.416,155.764
C08786=1051.176,-96.117,-67.784,170.122,30.417,155.764
C08787=1051.183,-95.868,-67.794,170.124,30.417,155.764
C08788=1051.189,-95.617,-67.805,170.126,30.418,155.764
C08789=1051.195,-95.368,-67.815,170.128,30.419,155.764
C08790=1051.201,-95.118,-67.826,170.131,30.420,155.764
C08791=1051.206,-94.868,-67.836,170.133,30.421,155.764
C08792=1051.213,-94.619,-67.846,170.135,30.422,155.764
C08793=1051.219,-94.369,-67.857,170.137,30.422,155.764
C08794=1051.225,-94.119,-67.867,170.138,30.423,155.764
C08795=1051.231,-93.869,-67.878,170.140,30.424,155.764
C08796=1051.237,-93.620,-67.889,170.143,30.425,155.764
C08797=1051.244,-93.370,-67.899,170.145,30.426,155.764
C08798=1051.249,-93.120,-67.910,170.147,30.427,155.764
C08799=1051.256,-92.871,-67.920,170.149,30.428,155.764
C08800=1051.261,-92.621,-67.931,170.151,30.429,155.764
C08801=1051.268,-92.371,-67.942,170.153,30.430,155.764
C08802=1051.274,-92.122,-67.952,170.156,30.431,155.764
C08803=1051.280,-91.872,-67.962,170.157,30.432,155.764
C08804=1051.285,-91.622,-67.973,170.159,30.433,155.764
C08805=1051.293,-91.372,-67.984,170.161,30.434,155.764
C08806=1051.298,-91.123,-67.995,170.163,30.434,155.764
C08807=1051.304,-90.873,-68.006,170.165,30.435,155.764
C08808=1051.311,-90.623,-68.016,170.168,30.436,155.764
C08809=1051.317,-90.373,-68.027,170.170,30.437,155.764
C08810=1051.323,-90.124,-68.037,170.172,30.438,155.764
C08811=1051.329,-89.874,-68.048,170.174,30.439,155.764
C08812=1051.335,-89.625,-68.059,170.175,30.440,155.764
C08813=1051.342,-89.375,-68.069,170.177,30.441,155.764
C08814=1051.348,-89.125,-68.080,170.180,30.442,155.764
C08815=1051.353,-88.875,-68.091,170.182,30.443,155.764
C08816=1051.360,-88.626,-68.101,170.184,30.444,155.764
C08817=1051.366,-88.376,-68.112,170.186,30.445,155.764
C08818=1051.372,-88.126,-68.123,170.188,30.445,155.764
C08819=1051.378,-87.877,-68.133,170.190,30.446,155.764
C08820=1051.385,-87.627,-68.145,170.193,30.447,155.764
C08821=1051.390,-87.377,-68.155,170.194,30.448,155.764
C08822=1051.397,-87.128,-68.166,170.196,30.449,155.765
C08823=1051.403,-86.878,-68.177,170.198,30.450,155.765
C08824=1051.409,-86.629,-68.188,170.200,30.451,155.765
C08825=1051.416,-86.379,-68.198,170.202,30.452,155.765
C08826=1051.422,-86.129,-68.209,170.204,30.453,155.765
C08827=1051.428,-85.880,-68.220,170.207,30.454,155.765
C08828=1051.435,-85.630,-68.231,170.209,30.455,155.765
C08829=1051.440,-85.380,-68.242,170.211,30.456,155.765
C08830=1051.447,-85.130,-68.253,170.212,30.457,155.765
C08831=1051.453,-84.881,-68.263,170.214,30.458,155.765
C08832=1051.459,-84.631,-68.274,170.216,30.459,155.765
C08833=1051.465,-84.381,-68.285,170.219,30.460,155.765
C08834=1051.471,-84.132,-68.296,170.221,30.461,155.765
C08835=1051.478,-83.882,-68.307,170.223,30.462,155.765
C08836=1051.484,-83.632,-68.318,170.225,30.463,155.765
C08837=1051.491,-83.348,-68.330,170.227,30.464,155.765
C08838=1051.498,-83.064,-68.343,170.230,30.465,155.765
C08839=1051.506,-82.781,-68.355,170.231,30.466,155.765
C08840=1051.513,-82.497,-68.368,170.234,30.467,155.765
C08841=1051.518,-82.247,-68.379,170.236,30.468,155.765
C08842=1051.525,-81.997,-68.390,170.238,30.469,155.765
C08843=1051.531,-81.748,-68.400,170.240,30.470,155.765
C08844=1051.538,-81.498,-68.411,170.242,30.471,155.766
C08845=1051.543,-81.248,-68.422,170.244,30.472,155.766
C08846=1051.550,-80.998,-68.434,170.247,30.473,155.766
C08847=1051.556,-80.749,-68.444,170.249,30.474,155.766
C08848=1051.563,-80.499,-68.456,170.250,30.475,155.766
C08849=1051.569,-80.250,-68.467,170.252,30.477,155.766
C08850=1051.576,-80.000,-68.477,170.254,30.478,155.766
C08851=1051.581,-79.750,-68.488,170.256,30.479,155.766
C08852=1051.588,-79.500,-68.499,170.258,30.480,155.766
C08853=1051.594,-79.251,-68.511,170.261,30.481,155.766
C08854=1051.600,-79.001,-68.522,170.263,30.482,155.766
C08855=1051.606,-78.752,-68.533,170.265,30.483,155.766
C08856=1051.612,-78.501,-68.544,170.266,30.484,155.766
C08857=1051.618,-78.252,-68.556,170.268,30.485,155.766
C08858=1051.625,-78.002,-68.567,170.270,30.486,155.766
C08859=1051.630,-77.753,-68.578,170.272,30.488,155.766
C08860=1051.637,-77.503,-68.589,170.274,30.489,155.767
C08861=1051.643,-77.254,-68.601,170.277,30.490,155.767
C08862=1051.649,-77.004,-68.612,170.279,30.491,155.767
C08863=1051.655,-76.754,-68.623,170.281,30.492,155.767
C08864=1051.661,-76.504,-68.635,170.282,30.493,155.767
C08865=1051.667,-76.255,-68.646,170.284,30.494,155.767
C08866=1051.674,-76.005,-68.657,170.286,30.496,155.767
C08867=1051.680,-75.755,-68.668,170.288,30.497,155.767
C08868=1051.686,-75.506,-68.680,170.290,30.497,155.767
C08869=1051.692,-75.256,-68.691,170.293,30.499,155.767
C08870=1051.698,-75.007,-68.703,170.295,30.500,155.767
C08871=1051.705,-74.756,-68.714,170.297,30.501,155.767
C08872=1051.710,-74.507,-68.725,170.298,30.502,155.767
C08873=1051.717,-74.257,-68.737,170.300,30.504,155.767
C08874=1051.723,-74.007,-68.748,170.302,30.505,155.768
C08875=1051.729,-73.758,-68.759,170.304,30.506,155.768
C08876=1051.736,-73.508,-68.771,170.306,30.507,155.768
C08877=1051.741,-73.259,-68.782,170.308,30.508,155.768
C08878=1051.748,-73.009,-68.794,170.311,30.510,155.768
C08879=1051.753,-72.759,-68.805,170.313,30.511,155.768
C08880=1051.760,-72.510,-68.817,170.314,30.512,155.768
C08881=1051.766,-72.260,-68.828,170.316,30.513,155.768
C08882=1051.772,-72.011,-68.840,170.318,30.515,155.768
C08883=1051.777,-71.761,-68.852,170.320,30.516,155.768
C08884=1051.784,-71.511,-68.864,170.322,30.517,155.769
C08885=1051.790,-71.261,-68.875,170.324,30.518,155.769
C08886=1051.796,-71.012,-68.886,170.326,30.520,155.769
C08887=1051.803,-70.762,-68.898,170.328,30.521,155.769
C08888=1051.808,-70.513,-68.910,170.329,30.522,155.769
C08889=1051.814,-70.263,-68.921,170.332,30.524,155.769
C08890=1051.821,-70.013,-68.933,170.334,30.525,155.769
C08891=1051.827,-69.764,-68.944,170.336,30.526,155.769
C08892=1051.832,-69.514,-68.956,170.338,30.527,155.769
C08893=1051.838,-69.264,-68.967,170.340,30.529,155.769
C08894=1051.845,-69.015,-68.979,170.342,30.530,155.770
C08895=1051.851,-68.765,-68.992,170.343,30.531,155.770
C08896=1051.857,-68.515,-69.003,170.345,30.532,155.770
C08897=1051.863,-68.266,-69.015,170.347,30.534,155.770
C08898=1051.869,-68.016,-69.026,170.349,30.535,155.770
C08899=1051.875,-67.766,-69.038,170.351,30.536,155.770
C08900=1051.881,-67.517,-69.050,170.353,30.538,155.770
C08901=1051.888,-67.235,-69.063,170.356,30.539,155.770
C08902=1051.895,-66.953,-69.076,170.358,30.541,155.770
C08903=1051.902,-66.672,-69.089,170.360,30.542,155.771
C08904=1051.909,-66.390,-69.103,170.362,30.544,155.771
C08905=1051.915,-66.139,-69.114,170.364,30.545,155.771
C08906=1051.921,-65.891,-69.126,170.366,30.546,155.771
C08907=1051.927,-65.641,-69.138,170.368,30.547,155.771
C08908=1051.934,-65.391,-69.150,170.370,30.549,155.771
C08909=1051.940,-65.142,-69.161,170.372,30.551,155.771
C08910=1051.945,-64.892,-69.174,170.373,30.551,155.771
C08911=1051.952,-64.642,-69.186,170.375,30.553,155.771
C08912=1051.958,-64.392,-69.197,170.378,30.554,155.771
C08913=1051.964,-64.143,-69.209,170.380,30.556,155.772
C08914=1051.970,-63.893,-69.221,170.382,30.557,155.772
C08915=1051.977,-63.644,-69.233,170.384,30.558,155.772
C08916=1051.983,-63.394,-69.244,170.386,30.560,155.772
C08917=1051.989,-63.144,-69.256,170.388,30.561,155.772
C08918=1051.995,-62.895,-69.268,170.389,30.562,155.772
C08919=1052.002,-62.645,-69.280,170.391,30.564,155.772
C08920=1052.007,-62.395,-69.292,170.393,30.565,155.773
C08921=1052.014,-62.146,-69.304,170.395,30.566,155.773
C08922=1052.020,-61.896,-69.316,170.397,30.568,155.773
C08923=1052.026,-61.646,-69.328,170.399,30.569,155.773
C08924=1052.033,-61.397,-69.340,170.401,30.570,155.773
C08925=1052.039,-61.147,-69.351,170.402,30.572,155.773
C08926=1052.045,-60.897,-69.364,170.405,30.573,155.773
C08927=1052.051,-60.648,-69.376,170.407,30.575,155.773
C08928=1052.058,-60.398,-69.388,170.409,30.576,155.773
C08929=1052.064,-60.148,-69.400,170.411,30.577,155.773
C08930=1052.070,-59.900,-69.412,170.413,30.579,155.774
C08931=1052.076,-59.650,-69.424,170.415,30.580,155.774
C08932=1052.082,-59.399,-69.436,170.417,30.582,155.774
C08933=1052.089,-59.150,-69.447,170.418,30.583,155.774
C08934=1052.095,-58.900,-69.460,170.420,30.584,155.774
C08935=1052.101,-58.651,-69.472,170.422,30.586,155.774
C08936=1052.107,-58.402,-69.484,170.424,30.587,155.774
C08937=1052.113,-58.152,-69.496,170.426,30.588,155.775
C08938=1052.120,-57.902,-69.508,170.428,30.590,155.775
C08939=1052.126,-57.653,-69.520,170.430,30.591,155.775
C08940=1052.132,-57.403,-69.533,170.431,30.592,155.775
C08941=1052.139,-57.153,-69.545,170.433,30.594,155.775
C08942=1052.144,-56.904,-69.557,170.436,30.596,155.775
C08943=1052.151,-56.654,-69.569,170.438,30.597,155.775
C08944=1052.158,-56.405,-69.581,170.440,30.598,155.775
C08945=1052.164,-56.155,-69.593,170.442,30.600,155.776
C08946=1052.170,-55.905,-69.605,170.444,30.601,155.776
C08947=1052.177,-55.656,-69.617,170.446,30.602,155.776
C08948=1052.183,-55.406,-69.630,170.447,30.604,155.776
C08949=1052.189,-55.156,-69.642,170.449,30.605,155.776
C08950=1052.195,-54.906,-69.654,170.451,30.606,155.776
C08951=1052.202,-54.657,-69.666,170.453,30.608,155.776
C08952=1052.208,-54.408,-69.678,170.455,30.609,155.776
C08953=1052.214,-54.158,-69.690,170.457,30.611,155.777
C08954=1052.221,-53.908,-69.702,170.459,30.612,155.777
C08955=1052.226,-53.659,-69.715,170.460,30.613,155.777
C08956=1052.233,-53.409,-69.727,170.462,30.615,155.777
C08957=1052.240,-53.159,-69.739,170.464,30.616,155.777
C08958=1052.246,-52.910,-69.751,170.466,30.617,155.777
C08959=1052.252,-52.660,-69.763,170.468,30.619,155.777
C08960=1052.258,-52.410,-69.776,170.470,30.620,155.778
C08961=1052.265,-52.161,-69.788,170.472,30.622,155.778
C08962=1052.271,-51.911,-69.800,170.474,30.624,155.778
C08963=1052.278,-51.662,-69.813,170.476,30.625,155.778
C08964=1052.284,-51.412,-69.825,170.478,30.626,155.778
C08965=1052.291,-51.131,-69.839,170.480,30.628,155.778
C08966=1052.299,-50.851,-69.852,170.482,30.629,155.778
C08967=1052.305,-50.570,-69.867,170.484,30.631,155.779
C08968=1052.312,-50.290,-69.881,170.487,30.633,155.779
C08969=1052.319,-50.040,-69.893,170.488,30.634,155.779
C08970=1052.325,-49.791,-69.906,170.490,30.636,155.779
C08971=1052.331,-49.541,-69.918,170.492,30.637,155.779
C08972=1052.337,-49.291,-69.931,170.494,30.639,155.779
C08973=1052.343,-49.042,-69.943,170.496,30.640,155.779
C08974=1052.349,-48.793,-69.956,170.498,30.642,155.780
C08975=1052.355,-48.543,-69.968,170.500,30.643,155.780
C08976=1052.361,-48.293,-69.981,170.501,30.645,155.780
C08977=1052.368,-48.044,-69.993,170.503,30.646,155.780
C08978=1052.374,-47.794,-70.006,170.505,30.648,155.780
C08979=1052.380,-47.544,-70.019,170.507,30.650,155.780
C08980=1052.386,-47.295,-70.031,170.509,30.651,155.781
C08981=1052.392,-47.046,-70.044,170.511,30.653,155.781
C08982=1052.398,-46.796,-70.056,170.513,30.655,155.781
C08983=1052.404,-46.546,-70.069,170.514,30.656,155.781
C08984=1052.411,-46.297,-70.082,170.516,30.658,155.781
C08985=1052.417,-46.047,-70.094,170.518,30.659,155.781
C08986=1052.423,-45.797,-70.107,170.520,30.661,155.782
C08987=1052.429,-45.548,-70.120,170.522,30.663,155.782
C08988=1052.435,-45.298,-70.133,170.524,30.664,155.782
C08989=1052.442,-45.048,-70.145,170.526,30.666,155.782
C08990=1052.448,-44.799,-70.158,170.527,30.667,155.782
C08991=1052.454,-44.549,-70.170,170.529,30.669,155.782
C08992=1052.460,-44.300,-70.184,170.531,30.670,155.783
C08993=1052.466,-44.050,-70.196,170.533,30.672,155.783
C08994=1052.473,-43.800,-70.208,170.535,30.673,155.783
C08995=1052.479,-43.551,-70.221,170.537,30.675,155.783
C08996=1052.485,-43.301,-70.234,170.539,30.676,155.783
C08997=1052.492,-43.051,-70.248,170.540,30.678,155.783
C08998=1052.498,-42.801,-70.260,170.542,30.680,155.784
C08999=1052.505,-42.553,-70.273,170.544,30.682,155.784
C09000=1052.510,-42.303,-70.285,170.546,30.683,155.784
C09001=1052.516,-42.053,-70.298,170.548,30.685,155.784
C09002=1052.523,-41.804,-70.311,170.550,30.686,155.784
C09003=1052.528,-41.554,-70.324,170.552,30.688,155.785
C09004=1052.535,-41.305,-70.337,170.553,30.689,155.785
C09005=1052.541,-41.055,-70.349,170.555,30.691,155.785
C09006=1052.548,-40.806,-70.362,170.557,30.693,155.785
C09007=1052.553,-40.556,-70.375,170.559,30.694,155.785
C09008=1052.560,-40.306,-70.389,170.561,30.696,155.785
C09009=1052.566,-40.056,-70.401,170.563,30.698,155.786
C09010=1052.573,-39.807,-70.414,170.565,30.699,155.786
C09011=1052.579,-39.558,-70.427,170.566,30.701,155.786
C09012=1052.585,-39.308,-70.440,170.568,30.702,155.786
C09013=1052.591,-39.058,-70.453,170.570,30.704,155.786
C09014=1052.597,-38.809,-70.465,170.572,30.705,155.786
C09015=1052.604,-38.559,-70.479,170.574,30.707,155.787
C09016=1052.610,-38.309,-70.492,170.576,30.709,155.787
C09017=1052.616,-38.059,-70.505,170.578,30.711,155.787
C09018=1052.623,-37.810,-70.518,170.579,30.712,155.787
C09019=1052.628,-37.560,-70.531,170.581,30.714,155.787
C09020=1052.635,-37.311,-70.544,170.583,30.716,155.788
C09021=1052.641,-37.062,-70.557,170.584,30.717,155.788
C09022=1052.647,-36.812,-70.570,170.586,30.719,155.788
C09023=1052.653,-36.563,-70.583,170.588,30.720,155.788
C09024=1052.660,-36.313,-70.597,170.590,30.723,155.788
C09025=1052.666,-36.063,-70.609,170.591,30.724,155.789
C09026=1052.672,-35.814,-70.623,170.593,30.726,155.789
C09027=1052.678,-35.564,-70.636,170.595,30.728,155.789
C09028=1052.684,-35.314,-70.648,170.597,30.729,155.789
C09029=1052.691,-35.034,-70.663,170.599,30.731,155.789
C09030=1052.697,-34.754,-70.678,170.602,30.733,155.790
C09031=1052.705,-34.474,-70.693,170.603,30.735,155.790
C09032=1052.712,-34.194,-70.708,170.605,30.737,155.790
C09033=1052.718,-33.944,-70.721,170.607,30.738,155.790
C09034=1052.724,-33.695,-70.735,170.609,30.741,155.790
C09035=1052.730,-33.446,-70.748,170.611,30.742,155.791
C09036=1052.737,-33.195,-70.761,170.613,30.744,155.791
C09037=1052.743,-32.946,-70.774,170.615,30.746,155.791
C09038=1052.749,-32.697,-70.787,170.616,30.747,155.791
C09039=1052.755,-32.448,-70.801,170.618,30.749,155.791
C09040=1052.761,-32.198,-70.813,170.620,30.751,155.792
C09041=1052.768,-31.948,-70.827,170.622,30.753,155.792
C09042=1052.774,-31.698,-70.841,170.624,30.754,155.792
C09043=1052.780,-31.449,-70.854,170.625,30.756,155.792
C09044=1052.786,-31.200,-70.867,170.627,30.758,155.792
C09045=1052.793,-30.950,-70.881,170.628,30.759,155.793
C09046=1052.799,-30.700,-70.893,170.630,30.761,155.793
C09047=1052.805,-30.450,-70.907,170.632,30.763,155.793
C09048=1052.811,-30.201,-70.920,170.634,30.764,155.793
C09049=1052.818,-29.951,-70.934,170.636,30.767,155.794
C09050=1052.824,-29.702,-70.947,170.638,30.768,155.794
C09051=1052.830,-29.452,-70.961,170.640,30.770,155.794
C09052=1052.836,-29.203,-70.974,170.641,30.772,155.794
C09053=1052.843,-28.953,-70.988,170.643,30.773,155.794
C09054=1052.849,-28.703,-71.000,170.645,30.775,155.794
C09055=1052.855,-28.454,-71.013,170.647,30.777,155.795
C09056=1052.862,-28.204,-71.027,170.649,30.779,155.795
C09057=1052.868,-27.955,-71.040,170.651,30.780,155.795
C09058=1052.874,-27.706,-71.054,170.652,30.782,155.795
C09059=1052.880,-27.455,-71.068,170.653,30.784,155.796
C09060=1052.886,-27.206,-71.081,170.655,30.785,155.796
